# B&R Automation Studio project AriesV2
Automation Studio 4.2.7.54 SP; technology packages: mapp 1.60.1, TextSystem 

## Configuration Config_3500HS

CPU X20CP1301, AutomationRuntime D4.24, Build 4.1.2, Vc V4.24.1, Safety 1.9

### Task classes (Cpu.sw)
```
Cyclic#1 (cycle 2000 us, tolerance 0 us):
  runFirst <- Libraries.wbrServices.InitSP.runFirst.prg (BuildOptions=-D "str(x)=#x" -D AS_PROJ=str($(AS_PROJECT_NAME)) -D AS_CFG=str($(AS_CONFIGURATION)) -D "AS_VERS=str($(AS_VERSION))" -D "AS_USER=str($(AS_USER_NAME))" -D "AS_CMPNY=str($(AS_COMPANY_NAME))")
  ForceIO1 <- HMI.ForceIO.prg
  ControlLog <- Application.Master.ControlLogic.prg
  Valves <- Application.Dispense.Valves.prg
  ForceIO <- HMI.ForceIO.prg
Cyclic#8 (cycle 24000 us, tolerance 48000 us):
  wbrService <- Libraries.wbrServices.Cyclic.wbrService.prg
  HMITableMa <- HMI.HMITableManager.prg
  Recipe_Han <- Auxiliary_Services_Control.Recipe_Handling.prg  // Call functions that manage structures pertaining to params
  hmilogic <- HMI.hmilogic.prg
  ComLogger <- Auxiliary_Services_Control.ComLogger.prg [disabled]
  File_Handl <- Auxiliary_Services_Control.File_Handling.prg
DataObjects: ethIPcon
VcDataObjects: VisuW1 <- HMI.VisuW1.dob
Binaries: TCData, vccpwd, vccbtn, vcpdvnc, arialbd, vcmgr, vctcal, vcfile, vccnum, vcfntttf, vcgclass, vcbclass, vccshape, vccstr, vccalarm, vccscale, arial, vcalarm, vcdsloc, vcchtml, vccdt, vccbmp, vcshared, vcxml, vccurl, vcrt, vcctext, vcnet, vcclbox, vcdsint, vcpdsw, vccovl, vccline, VisuW101, VisuW102, VisuW103, vera, vccgauge, vcpfx20, TC, Data_Log, MAPP_Alm, MAPP_Rec, MAPP_Web, MAPP_File, MAPP_Cfg, iomap, asfw, sysconf, ashwd, arconfig, Alarm, vcctrend, vccpopup, vccddbox, vccpiech, vcpkat, verabd, Visu, Visu02, Visu03, Visu01, Axes, Config_1, MAPP_Com, Recipe, File_Mgmt, vccslider, Acp10Map1, User, Role, Data, Config, VisuW03, VisuW02, VisuW01, acp10cfg, Acp10map, Acp10sys, vcpfar00
Libraries: wbrsprintf, FileIO, AsXml, standard, runtime, astime, brsystem, sys_lib, AsANSL, AsARCfg, AsBrMath, AsBrStr, DataObj, AsTCP, AsUDP, AsUSB, MpCom, MpAlarm, MpFile, MpRecipe, MpWebXs, AsArSdm, AsIecCon, operator, AsIOTime, AsMem, AsArLog, AsArProf, MTBasics, MTTypes, MTFilter, jgLibC, MTData, ArTextSys, AsICMP, bglibasWBR, MAPPSuppor, wbrFltUtil, wbrListSvc, wbrLogSvc, wbrMemSvc, wbrPingSvc, libValve, libAS52XX, vcresman, arsvcreg, ashw, AsMbTCP, AsSafety, powerlnk
```

### Hardware
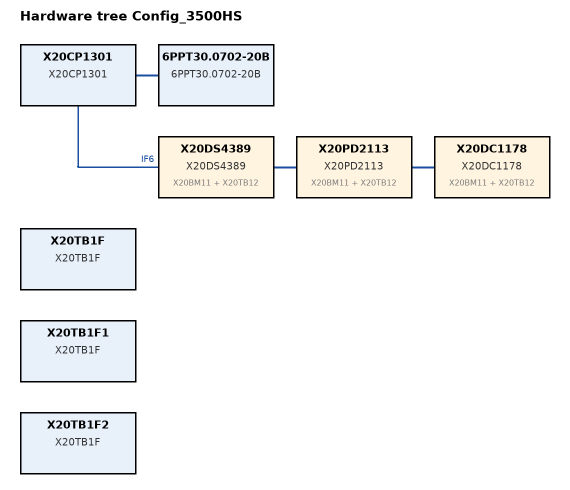
```
6PPT30.0702-20B : 6PPT30.0702-20B v1.1.0.0 (LastFrozenVersion=1.1.0.0)  [ETH1 -> X20CP1301.IF2 (NodeNumber=1)]
  Terminal = true
  Startmode = 1
  Mode = Manual
  InternetAddress = 192.168.10.20
  DefaultGateway = 192.168.10.10
  Subnetmask = 255.255.255.0
  Hostname = t30_panel
  Displaybrightness = 90
  SelectedFavoriteVNC = 192.168.10.10:5900
  PasswordVNC = 
  Favorites_Web1 = 192.168.10.10/SDM
  Favorites_Web2 = 192.168.10.10/MAPP
  USBmemoryshare = 0
  Usermemoryshare = 0
  PasswordCIFS = 
  PasswordService = 
  PPTImage = PPT_30_V1.1.0
  VncVcObjectName = VisuW1
  VncKeyMappingFile = VC\6PPT30.070.dis
  VncMaxConnections = 2
  VncRefreshRate = 300
X20BM11 : X20BM11 v1.0.0.0  [X2X1 -> X20CP1301.IF6]
X20BM11a : X20BM11 v1.0.0.0  [X2X1 -> X20BM11.X2X2]
X20BM11b : X20BM11 v1.0.0.0  [X2X1 -> X20BM11a.X2X2]
X20CP1301 : X20CP1301 v1.0.4.0  [X1 -> X1.SL; X2 -> X2.SL; X3 -> X3.SL]
  Module X1 (Type=X1, Virtual=true, Version=1.0.0.0)
    Connection (Connector=SS1, TargetModule=X20TB1F, TargetConnector=SS)
    Connection (Connector=SL, TargetModule=X20CP1301, TargetConnector=X1)
  Module X2 (Type=X2, Virtual=true, Version=1.0.0.0)
    Connection (Connector=SS1, TargetModule=X20TB1F1, TargetConnector=SS)
    Connection (Connector=SL, TargetModule=X20CP1301, TargetConnector=X2)
  Module X3 (Type=X3, Virtual=true, Version=1.0.0.0)
    Connection (Connector=SS1, TargetModule=X20TB1F2, TargetConnector=SS)
    Connection (Connector=SL, TargetModule=X20CP1301, TargetConnector=X3)
  Connector IF2:
    ActivateDevice = 1
    HostName = cp1382
    Mode = Manual
    InternetAddress = 192.168.10.10
    SubnetMask = 255.255.255.0
    InaNodeNumber = 1
  Connector IF6:
    CycleTime = 1000
  UserRamSize = 9000
  RemMemSize = 6000
  PermanentPvSize = 6000
  VolatileGlobalPvSize = 200000
  RebootPowerfail = 2
  TimerDeviceType = SWIOTIMER
  TaskClassIdleTime = 8000
  Cyclic1Duration = 2000
  Cyclic1Tolerance = 0
  Cyclic1Input = 1
  Cyclic1Output = 1
  Cyclic2Duration = 10000
  Cyclic2Tolerance = 1000000
  Cyclic3Duration = 10000
  Cyclic3Tolerance = 5000000
  Cyclic4Duration = 100000
  Cyclic4Tolerance = 100000
  Cyclic5Duration = 200000
  Cyclic5Tolerance = 200000
  Cyclic6Duration = 500000
  Cyclic6Tolerance = 500000
  Cyclic7Duration = 1000000
  Cyclic7Tolerance = 1000000
  Cyclic8Duration = 24000
  Cyclic8Tolerance = 48000
  FileDevice1
  FileDeviceName1 = ROOT
  FileDevicePath1 = F:\
  FileDevice2
  FileDeviceName2 = Recipe
  FileDevicePath2 = F:\AS_Data\Recipe
  FileDevice3
  FileDeviceName3 = Config
  FileDevicePath3 = F:\AS_Data\Config
  FtpUser1
  FtpUsername1 = user
  FtpUserPassword1 = LsodGR3jeFK3pzrFw1H5+czzepg0YTVl3svctHEKl8w=
  FtpUserSalt1 = HHFLDaL4
  FTPAccessRight1 = 0
  FtpUser2
  FtpUsername2 = admin
  FtpUserPassword2 = ohx/+BSKxELE8VtAzHGH48r+NF8pZu2EVGO55B1GtgA=
  FtpUserSalt2 = HlYZIA1j
  FTPPath2 = 5
  FTPAccessRight2 = 0
  SystemTick = 2000
X20DC1178 : X20DC1178 v1.0.0.1  [SS1 -> X20TB12b.SS; SL -> X20BM11b.SL1]
  Supervision = off
  CounterStd01 = 16Bit
  ClockrateSSI = 125kHz
  DataFormatSSI = gray
  ValidBitLengthSSI = 12
  CycleSelect = 50us
  MonoflopSSI = HIGH
  BrokenWireConfig = off
X20DS4389 : X20DS4389 v1.2.0.0  [SS1 -> X20TB12a.SS; SL -> X20BM11.SL1]
  Supervision = off
  Channel01Config = inputInv
  Channel02Config = inputInv
  Channel03Config = outputPush
  Channel04Config = outputPush
  Channel05Config = inputInv
  Channel06Config = inputInv
  Channel07Config = outputPush
  Channel08Config = outputPush
  DirectIOControlConfig = on
  EdgeDetectEnable = on
  EdgeDetectUnit01Master = 2
  EdgeDetectUnit01Slave = 18
  EdgeDetectUnit01EnableDifference = 32bit
  EdgeDetectUnit02Master = 18
  EdgeDetectUnit02Slave = 2
  EdgeDetectUnit02EnableDifference = 32bit
  EdgeDetectUnit03Master = 3
  EdgeDetectUnit03Slave = 19
  EdgeDetectUnit03EnableDifference = 32bit
  EdgeDetectUnit04Master = 19
  EdgeDetectUnit04Slave = 3
  EdgeDetectUnit04EnableDifference = 32bit
  EdgeGenerateEnable = on
  EdgeGenOutputUpdateCycle = SOAIEOP
  EdgeGenerateUnit01Enable = on
  EdgeGenUnit01TimeStamps = 1elem
  EdgeGenUnit01TimeFormat = 32bit
  EdgeGenUnit01OffsetFormat = 32bit
  EdgeGenUnit01OffsetFormat01 = cyclic
  EdgeGenUnit01Edge01Enable = on
  EdgeGenUnit01Edge01Channel = 2
  EdgeGenUnit01Edge02Enable = on
  EdgeGenerateUnit02Enable = on
  EdgeGenUnit02TimeStamps = 1elem
  EdgeGenUnit02TimeFormat = 32bit
  EdgeGenUnit02OffsetFormat = 32bit
  EdgeGenUnit02OffsetFormat01 = cyclic
  EdgeGenUnit02Edge01Enable = on
  EdgeGenUnit02Edge01Channel = 3
  EdgeGenUnit02Edge02Enable = on
  EdgeGenUnit01Edge02Channel = 18
  EdgeGenUnit02Edge02Channel = 19
  DirectIOInputs = on
X20PD2113 : X20PD2113 v1.0.2.0  [SS1 -> X20TB12.SS; SL -> X20BM11a.SL1]
X20TB12 : X20TB12 v1.0.0.0
X20TB12a : X20TB12 v1.0.0.0
X20TB12b : X20TB12 v1.0.0.0
X20TB1F : X20TB1F v1.0.0.0
X20TB1F1 : X20TB1F v1.0.0.0
X20TB1F2 : X20TB1F v1.0.0.0
```

### IoMap.iom - X20CP1301/IoMap.iom
```iecst
VAR_CONFIG
	Cyclic#1.ControlIO.iTargetPiP AT %IX."X1".DigitalInput01;
	Cyclic#1.ControlIO.iReservoirLevel AT %IX."X1".DigitalInput02;
	Cyclic#1.ControlIO.iRunCmd AT %IX."X1".DigitalInput03;
	Cyclic#1.StatusIO.iClearError AT %IX."X1".DigitalInput04;
	Cyclic#1.CureIO.iUVCuringChannelOK[0] AT %IX."X2".DigitalInput01;
	Cyclic#1.CureIO.iUVCuringChannelOK[1] AT %IX."X2".DigitalInput02;
	Cyclic#1.StatusIO.iProcessStopRelay[0] AT %IX."X2".DigitalInput03;
	Cyclic#1.StatusIO.iProcessStopRelay[1] AT %IX."X2".DigitalInput04;
	Cyclic#1.ControlIO.iX2XNettime AT %ID."X20CP1301".IF6.Nettime;
	Cyclic#1.ControlIO.iEncoderValue AT %IW."X20DC1178".Encoder01;
	Cyclic#1.StatusIO.Encoder.CycleTimeViolation.iErrorStatus AT %IX."X20DC1178".EncoderCycleTimeViolation;
	Cyclic#1.StatusIO.Encoder.DataError.iErrorStatus AT %IX."X20DC1178".EncoderDataError;
	Cyclic#1.StatusIO.Encoder.CycleTimeViolation.oQuitError AT %QX."X20DC1178".EncoderQuitCycleTimeViolation;
	Cyclic#1.StatusIO.Encoder.DataError.oQuitError AT %QX."X20DC1178".EncoderQuitDataError;
	Cyclic#1.StatusIO.Encoder.iPowerSupply[0] AT %IX."X20DC1178".PowerSupply01;
	Cyclic#1.StatusIO.Encoder.iPowerSupply[1] AT %IX."X20DC1178".PowerSupply02;
	Cyclic#1.ValveIO[0].iValveReady AT %IX."X20DS4389".DigitalInput01 INVERSE;
	Cyclic#1.ValveIO[1].iValveReady AT %IX."X20DS4389".DigitalInput02 INVERSE;
	Cyclic#1.ValveIO[0].EdgeGen.iDiffTime[0] AT %ID."X20DS4389".EdgeDetect01Difference1;
	Cyclic#1.ValveIO[0].EdgeGen.iDiffTime[1] AT %ID."X20DS4389".EdgeDetect02Difference1;
	Cyclic#1.ValveIO[0].EdgeGen.oEnableEdgeGen AT %QX."X20DS4389".EdgeGen01Enable;
	Cyclic#1.ValveIO[0].EdgeGen.iEdgeGenReadbackEnabled AT %IX."X20DS4389".EdgeGen01EnableReadback;
	Cyclic#1.ValveIO[0].EdgeGen.oEdgeGenOffset AT %QD."X20DS4389".EdgeGen01Offset1;
	Cyclic#1.ValveIO[0].EdgeGen.oEdgeGenSequence AT %QB."X20DS4389".EdgeGen01Sequence;
	Cyclic#1.ValveIO[0].EdgeGen.oEdgeGenTimestamp AT %QD."X20DS4389".EdgeGen01Timestamp1;
	Cyclic#1.ValveIO[1].EdgeGen.oEnableEdgeGen AT %QX."X20DS4389".EdgeGen02Enable;
	Cyclic#1.ValveIO[1].EdgeGen.iEdgeGenReadbackEnabled AT %IX."X20DS4389".EdgeGen02EnableReadback;
	Cyclic#1.ValveIO[1].EdgeGen.oEdgeGenOffset AT %QD."X20DS4389".EdgeGen02Offset1;
	Cyclic#1.ValveIO[1].EdgeGen.oEdgeGenSequence AT %QB."X20DS4389".EdgeGen02Sequence;
	Cyclic#1.ValveIO[1].EdgeGen.oEdgeGenTimestamp AT %QD."X20DS4389".EdgeGen02Timestamp1;
	Cyclic#1.CureIO.oUVCureChannel[0] AT %QX."X3".DigitalOutput01;
	Cyclic#1.CureIO.oUVCureChannel[1] AT %QX."X3".DigitalOutput02;
	Cyclic#1.StatusIO.oRunningReady AT %QX."X3".DigitalOutput04;
	Cyclic#1.StatusIO.oSystemNeedsAttention AT %QX."X3".DigitalOutput05;
	Cyclic#1.ControlIO.oTargetPresent AT %QX."X3".DigitalOutput06;
	Cyclic#1.ControlIO.Inspection.oInspectionGood AT %QX."X3".DigitalOutput07;
	Cyclic#1.ControlIO.Inspection.oInspectionValid AT %QX."X3".DigitalOutput08;
	Cyclic#1.StatusIO.oStatusColor.Red AT %QX."X3".DigitalOutput09;
	Cyclic#1.StatusIO.oStatusColor.Green AT %QX."X3".DigitalOutput10;
	Cyclic#1.StatusIO.oStatusColor.Blue AT %QX."X3".DigitalOutput11;
END_VAR
```

### Data_Log.mpdatarecorder - X20CP1301/mapp/Data_Log.mpdatarecorder
```
Element Data_Log_MpLink (Type=mpdatarecorder)
  DataRecorder:
    MaxNumberOfFiles = 15
    DecimalDigits = 3
    SaveInterval = 60000
    PowerFailSafe = FALSE
    DecimalMark = .
    OverwriteOldestFile = TRUE
```

## Configuration Config_Deployment

### Task classes (Cpu.sw)
```
Cyclic#1 (cycle 4000 us, tolerance 0 us):
  ForceIO <- HMI.ForceIO.prg
  Creaser <- Application.Creaser.prg
  ForceIO1 <- HMI.ForceIO.prg
Cyclic#8 (cycle 8000 us, tolerance 30000000 us):
  LineContro <- MotionControl.LineControl.prg
  HMI_Alarms <- HMI.HMI_Alarms.prg
  Recipe_Han <- Auxiliary_Services_Control.Recipe_Handling.prg
  hmilogic <- HMI.hmilogic.prg
  HMITableMa <- HMI.HMITableManager.prg
  File_Handl <- Auxiliary_Services_Control.File_Handling.prg
  ComLogger <- Auxiliary_Services_Control.ComLogger.prg
DataObjects: Acp10sys, ethIPcon
NcDataObjects: acp10etxen <- acp10etxen.dob, Axisa <- Axisobj.Axisa.dob, Axisi <- Axisobj.Axisi.dob
VcDataObjects: Visup <- HMI.Visup.dob
Binaries: vcfntttf, vccbmp, vcshared, vccscale, vcpdvnc, Visup01, vcfile, vccpwd, arial, Visup03, vcmgr, vcxml, vcdsint, vccbtn, vcdsloc, vccalarm, vccovl, vcpfx20, vccline, vcctext, vcalarm, vcbclass, vcgclass, udbdef, vcrt, vccnum, vccstr, vccddbox, arialbd, vera, vccshape, vcpdsw, vccpopup, Visup02, vccurl, vcnet, arsvcreg, TCData, vcchtml, vctcal, vccdt, vcpkat, vcclbox, Data_Log, MAPP_Alm, MAPP_Rec, Alarm, MAPP_Web, ashwd, arconfig, MAPP_File, Config, asfw, sysconf, TC, MAPP_Cfg, iomap, acp10cfg, Acp10map, vcpfar00, Visu102, Visu101, Visu103, VisuW101, vcctrend, vccpiech, verabd, Visu, Visu02, Visu03, Visu01, Axes, Config_1, MAPP_Com, Recipe, File_Mgmt, vccslider, Acp10Map1, User, Role, Data, VisuW03, VisuW02, VisuW01, vccgauge, VisuW103, VisuW102
Libraries: FileIO, AsXml, standard, runtime, astime, brsystem, sys_lib, AsANSL, AsARCfg, AsBrMath, AsBrStr, DataObj, AsTCP, AsUDP, AsUSB, AsArSdm, AsIecCon, operator, AsIOTime, AsMem, AsArLog, AsArProf, AsICMP, Acp10man, Acp10par, NcGlobal, Acp10_MC, MpAxis, MpCom, wbrsprintf, wbrPingSvc, wbrMemSvc, wbrLogSvc, wbrListSvc, wbrFltUtil, MpWebXs, MpRecipe, MpFile, MpAlarm, MAPPSuppor, jgLibC, bglibasWBR, Acp10sim, ArTextSys, vcresman, powerlnk, ashw, MTTypes, AsMbTCP, AsSafety, MTData
```

### Hardware
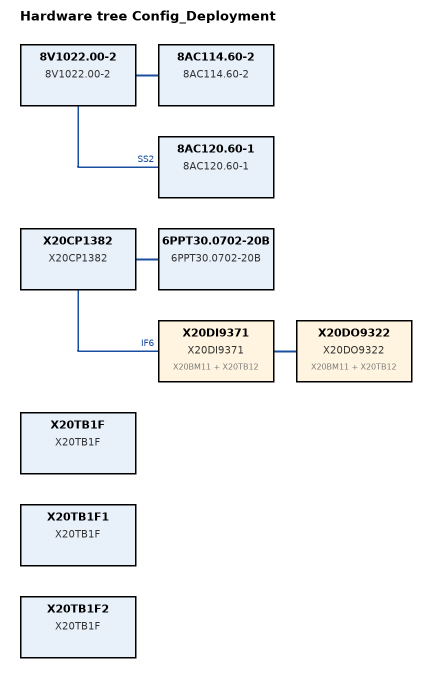
```
6PPT30.0702-20B : 6PPT30.0702-20B v1.1.0.0  [ETH1 -> X20CP1382.IF2 (NodeNumber=1)]
  Terminal = true
  Startmode = 1
  ShowBootlogoVNC = 1
  Mode = Manual
  InternetAddress = 192.168.10.20
  DefaultGateway = 192.168.10.1
  Subnetmask = 255.255.255.0
  Displaybrightness = 75
  SelectedFavoriteVNC = 192.168.10.10
  Favorites_VNC1 = 192.168.10.10
  PasswordVNC = 
  PasswordCIFS = 
  PasswordService = 
  PPTImage = PPT_30_V1.1.1
  VncRefreshRate = 200
8AC114.60-2 : 8AC114.60-2 v1.0.0.8  [SS -> 8V1022.00-2.SS1; PLK1 -> X20CP1382.IF3 (NodeNumber=2)]
8AC120.60-1 : 8AC120.60-1 v1.0.0.2  [SS -> 8V1022.00-2.SS2]
8V1022.00-2 : 8V1022.00-2 v1.0.0.2
  AxisIsPeriodic_r1 = on
  BothEndSwitchesAreNormallyOpen_r1 = on
  QuickStopIsNormallyOpen_r1 = on
X20BM11 : X20BM11 v1.0.0.1  [X2X1 -> X20CP1382.IF6]
X20BM11a : X20BM11 v1.0.0.1  [X2X1 -> X20BM11.X2X2]
X20CP1382 : X20CP1382 v1.3.2.0  [X1 -> X1.SL; X2 -> X2.SL; X3 -> X3.SL]
  Module X1 (Type=X1, Virtual=true, Version=1.0.0.0)
    Connection (Connector=SS1, TargetModule=X20TB1F, TargetConnector=SS)
    Connection (Connector=SL, TargetModule=X20CP1382, TargetConnector=X1)
  Module X2 (Type=X2, Virtual=true, Version=1.0.0.0)
    Connection (Connector=SS1, TargetModule=X20TB1F1, TargetConnector=SS)
    Connection (Connector=SL, TargetModule=X20CP1382, TargetConnector=X2)
  Module X3 (Type=X3, Virtual=true, Version=1.0.0.0)
    Connection (Connector=SS1, TargetModule=X20TB1F2, TargetConnector=SS)
    Connection (Connector=SL, TargetModule=X20CP1382, TargetConnector=X3)
  Connector IF2:
    ActivateDevice = 1
    HostName = x20cpu
    Mode = Manual
    InternetAddress = 192.168.10.10
    SubnetMask = 255.255.255.0
    InaNodeNumber = 0
    Vnc1
    VncVcObjectName1 = Visup
    VncKeyMappingFile1 = VC\PS2-Keyboard4.dis
    VncRefreshRate1 = 200
  Connector IF3:
    CycleTime = 4000
  Connector IF6:
    CycleTime = 4000
  ConfigurationID = AriesV2_Config_Test
  UserPartitionSize = 256
  UserRamSize = 5000
  RemMemSize = 25000
  PermanentPvSize = 15000
  VolatileGlobalPvSize = 300000
  RebootReset = 2
  RebootPowerfail = 2
  TimerDeviceType = EPLX2X
  TimerDevice = X20CP1382.IF3
  TaskClassIdleTime = 8000
  Cyclic1Duration = 4000
  Cyclic1Tolerance = 0
  Cyclic2Duration = 16000
  Cyclic2Tolerance = 16000
  Cyclic3Duration = 48000
  Cyclic3Tolerance = 48000
  Cyclic4Duration = 96000
  Cyclic4Tolerance = 96000
  Cyclic5Duration = 200000
  Cyclic5Tolerance = 200000
  Cyclic6Duration = 496000
  Cyclic6Tolerance = 496000
  Cyclic7Duration = 1000000
  Cyclic7Tolerance = 1000000
  Cyclic8Duration = 8000
  Cyclic8Tolerance = 30000000
  FileDevice1
  FileDeviceName1 = ROOT
  FileDevicePath1 = F:\
  FileDevice2
  FileDeviceName2 = Config
  FileDevicePath2 = F:\Config
  FileDevice3
  FileDeviceName3 = Recipe
  FileDevicePath3 = F:\Recipe
  FileDevice4
  FileDeviceName4 = Process
  FileDevicePath4 = F:\Process
  FtpUser1
  FtpUsername1 = admin
  FtpUserPassword1 = tXcQUdKIsoY/H/jtKSqzHLRzyWbO/eZFb+QmJVs8vuM=
  FtpUserSalt1 = fFlgpUU6
  FTPAccessRight1 = 0
  FTPdevice1 = ALL
  FtpUser2
  FtpUsername2 = user
  FtpUserPassword2 = M/sBBWLbPcMSL0ECBo9+NNWk5QFExAfaSSh+paOlJpQ=
  FtpUserSalt2 = diDYFxUT
  FTPAccessRight2 = 0
  FTPMSpath2 = /
X20DI9371 : X20DI9371 v1.0.1.3  [SS1 -> X20TB12.SS; SL -> X20BM11.SL1]
  Supervision = off
X20DO9322 : X20DO9322 v1.0.3.0  [SS1 -> X20TB12a.SS; SL -> X20BM11a.SL1]
  Supervision = off
X20TB12 : X20TB12 v1.0.0.0
X20TB12a : X20TB12 v1.0.0.0
X20TB1F : X20TB1F v1.0.0.0
X20TB1F1 : X20TB1F v1.0.0.0
X20TB1F2 : X20TB1F v1.0.0.0
```

### Config.mpaxisbasic - X20CP1382/mapp/Config.mpaxisbasic
```
Element FeedAxis_MpLink (Type=mpaxisbasic)
  AxisConfiguration = AxisWithConfiguration
    Axis:
      MeasurementUnit = 1
      MeasurementResolution = 0.001
      PeriodSettings:
        Period = 125.664
      MovementLimits:
        VelocityPositive = 10000.0
        VelocityNegative = 10000.0
        Acceleration = 10000.0
        Deceleration = 10000.0
        PositionErrorStopLimit = 1
    Drive:
      Gearbox:
        Input = 5
      Transformation:
        ReferenceDistance = 125.664
      Controller:
        Speed:
          ProportionalGain = 1.75
          IntegralTime = 1
        LoopFilters:
          [0]
          [1]
          [2]
```

## Configuration Config_Test

CPU X20CP1382, AutomationRuntime B4.26, Build 4.1.2, Vc V4.26.3, Safety 0.0

CPU X20CP1584, AutomationRuntime B4.26, Build 4.1.2, Vc not used, Safety 1.5

### Task classes (Cpu.sw)
```
Cyclic#1 (cycle 8000 us, tolerance 0 us):
  ForceIO <- HMI.ForceIO.prg [disabled]
  Creaser <- Application.Creaser.prg
  ForceIO1 <- HMI.ForceIO.prg [disabled]
DataObjects: ethIPcon
NcDataObjects: acp10etxen <- acp10etxen.dob, Axisa <- Axisobj.Axisa.dob, Axisi <- Axisobj.Axisi.dob
Binaries: TCData, Acp10sys, udbdef, Alarm, ashwd, asfw, MAPP_Cfg, MAPP_File, MAPP_Web, MAPP_Rec, MAPP_Alm, Data_Log, arconfig, sysconf, iomap, Config, acp10cfg, Acp10map, vcpdvnc, vcmgr, vctcal, vcnet, VisuW101, vcpfx20, vcctrend, vccpopup, vccddbox, vccpiech, vcpkat, verabd, Visu, Visu02, Visu03, Visu01, Axes, Config_1, MAPP_Com, Recipe, File_Mgmt, vccslider, Acp10Map1, User, Role, Data, VisuW03, VisuW02, VisuW01, vcpfar00, TC, vccgauge, vera, VisuW103, VisuW102, vccline, vccovl, vcpdsw, vcdsint, vcclbox, vcctext, vcrt, vccurl, vcxml, vcshared, vccbmp, vccdt, vcchtml, vcdsloc, vcalarm, arial, vccscale, vccalarm, vccstr, vccshape, vcbclass, vcgclass, vcfntttf, vccnum, vcfile, arialbd, vccbtn, vccpwd
Libraries: FileIO, AsXml, standard, runtime, astime, brsystem, sys_lib, AsANSL, AsARCfg, AsBrMath, AsBrStr, DataObj, AsTCP, AsUDP, AsUSB, AsArSdm, AsIecCon, operator, AsIOTime, AsMem, AsArLog, AsArProf, AsICMP, powerlnk, Acp10man, Acp10par, NcGlobal, Acp10_MC, MpAxis, MpCom, wbrsprintf, wbrPingSvc, wbrMemSvc, wbrLogSvc, wbrListSvc, wbrFltUtil, MpWebXs, MpRecipe, MpFile, MpAlarm, MAPPSuppor, jgLibC, bglibasWBR, arsvcreg, ashw, AsMbTCP, AsSafety, vcresman
```

### Task classes (Cpu.sw)
```
DataObjects: ethIPcon
Binaries: TCData, Alarm, ashwd, asfw, MAPP_Cfg, MAPP_File, MAPP_Web, MAPP_Rec, MAPP_Alm, Data_Log, arconfig, sysconf, iomap, vcpdvnc, vcmgr, vctcal, vcnet, VisuW101, vcpfx20, vcctrend, vccpopup, vccddbox, vccpiech, vcpkat, verabd, Visu, Visu02, Visu03, Visu01, Axes, Config_1, MAPP_Com, Recipe, File_Mgmt, vccslider, Acp10Map1, User, Role, Data, Config, VisuW03, VisuW02, VisuW01, acp10cfg, Acp10map, Acp10sys, vcpfar00, TC, vccgauge, vera, VisuW103, VisuW102, vccline, vccovl, vcpdsw, vcdsint, vcclbox, vcctext, vcrt, vccurl, vcxml, vcshared, vccbmp, vccdt, vcchtml, vcdsloc, vcalarm, arial, vccscale, vccalarm, vccstr, vccshape, vcbclass, vcgclass, vcfntttf, vccnum, vcfile, arialbd, vccbtn, vccpwd
Libraries: FileIO, AsXml, standard, runtime, astime, brsystem, sys_lib, AsANSL, AsARCfg, AsBrMath, AsBrStr, DataObj, AsTCP, AsUDP, AsUSB, AsArSdm, AsIecCon, operator, AsIOTime, AsMem, AsArLog, AsArProf, AsICMP, arsvcreg, ashw, AsMbTCP, AsSafety, powerlnk, vcresman
```

### Hardware
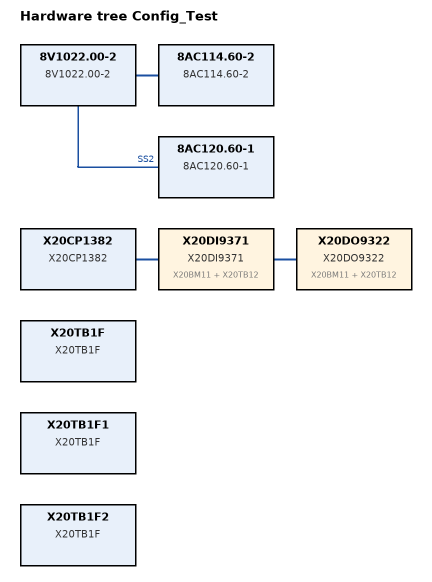
```
8AC114.60-2 : 8AC114.60-2 v1.0.0.8  [SS -> 8V1022.00-2.SS1; PLK1 -> X20CP1382.IF3 (NodeNumber=2)]
8AC120.60-1 : 8AC120.60-1 v1.0.0.2  [SS -> 8V1022.00-2.SS2]
8V1022.00-2 : 8V1022.00-2 v1.0.0.2
  AxisIsPeriodic_r1 = on
  BothEndSwitchesAreNormallyOpen_r1 = on
  QuickStopIsNormallyOpen_r1 = on
X20BM11 : X20BM11 v1.0.0.1  [X2X1 -> X20CP1382.IF6]
X20BM11a : X20BM11 v1.0.0.1  [X2X1 -> X20BM11.X2X2]
X20CP1382 : X20CP1382 v1.3.2.0  [X1 -> X1.SL; X2 -> X2.SL; X3 -> X3.SL]
  Module X1 (Type=X1, Virtual=true, Version=1.0.0.0)
    Connection (Connector=SS1, TargetModule=X20TB1F, TargetConnector=SS)
    Connection (Connector=SL, TargetModule=X20CP1382, TargetConnector=X1)
  Module X2 (Type=X2, Virtual=true, Version=1.0.0.0)
    Connection (Connector=SS1, TargetModule=X20TB1F1, TargetConnector=SS)
    Connection (Connector=SL, TargetModule=X20CP1382, TargetConnector=X2)
  Module X3 (Type=X3, Virtual=true, Version=1.0.0.0)
    Connection (Connector=SS1, TargetModule=X20TB1F2, TargetConnector=SS)
    Connection (Connector=SL, TargetModule=X20CP1382, TargetConnector=X3)
  Connector IF2:
    ActivateDevice = 1
    HostName = x20cpu
    Mode = Manual
    InternetAddress = 192.168.10.10
    SubnetMask = 255.255.255.0
    InaNodeNumber = 0
    Vnc1
    VncVcObjectName1 = Visu1
    VncKeyMappingFile1 = VC\PS2-Keyboard4.dis
    VncRefreshRate1 = 200
  Connector IF3:
    CycleTime = 8000
  Connector IF6:
    CycleTime = 8000
  ConfigurationID = AriesV2_Config_Test
  UserRamSize = 5000
  RemMemSize = 25000
  PermanentPvSize = 15000
  VolatileGlobalPvSize = 300000
  RebootReset = 2
  RebootPowerfail = 2
  TimerDeviceType = EPLX2X
  TimerDevice = X20CP1382.IF3
  TaskClassIdleTime = 8000
  Cyclic1Duration = 8000
  Cyclic1Tolerance = 0
  Cyclic2Duration = 16000
  Cyclic2Tolerance = 16000
  Cyclic3Duration = 48000
  Cyclic3Tolerance = 48000
  Cyclic4Duration = 96000
  Cyclic4Tolerance = 96000
  Cyclic5Duration = 200000
  Cyclic5Tolerance = 200000
  Cyclic6Duration = 496000
  Cyclic6Tolerance = 496000
  Cyclic7Duration = 1000000
  Cyclic7Tolerance = 1000000
  Cyclic8Duration = 8000
  Cyclic8Tolerance = 30000000
  FileDevice1
  FileDeviceName1 = ROOT
  FileDevicePath1 = F:\
  FileDevice2
  FileDeviceName2 = Config
  FileDevicePath2 = F:\Config
  FileDevice3
  FileDeviceName3 = Recipe
  FileDevicePath3 = F:\Recipe
  FileDevice4
  FileDeviceName4 = Process
  FileDevicePath4 = F:\Process
X20DI9371 : X20DI9371 v1.0.2.0  [SS1 -> X20TB12.SS; SL -> X20BM11.SL1]
  Supervision = off
X20DO9322 : X20DO9322 v1.0.3.0  [SS1 -> X20TB12a.SS; SL -> X20BM11a.SL1]
  Supervision = off
X20TB12 : X20TB12 v1.0.0.0
X20TB12a : X20TB12 v1.0.0.0
X20TB1F : X20TB1F v1.0.0.0
X20TB1F1 : X20TB1F v1.0.0.0
X20TB1F2 : X20TB1F v1.0.0.0
```

### Cpu.per - X20CP1382/Cpu.per
```iecst
VAR_CONFIG
	gRecipeName AT %M0; (* *)
	gConfigName AT %M256; (* *)
	gStatistics AT %M512; (* *)
	gRecCfg AT %M600; (* *)
END_VAR
```

### Acp10map.ncm - X20CP1584/Motion/Acp10map.ncm
```
NcMapping (NcSwId=Acp10)
  NcObject Axis (ModuleId=8V1045.00-2, Type=ncAXIS, Channel=1, AcoposSimulation=Off, InitParameter=Axisi, AcoposParameter=Axisa, AdditionalData=PLCopen_ModPos="1000,1" , Disabled=FALSE, ModuleDisabled=FALSE)
  NcObject 8V1045.00-2_ncV_AXIS1 (ModuleId=8V1045.00-2, Type=ncV_AXIS, Channel=1, Disabled=TRUE, ModuleDisabled=FALSE)
```

### Config.mpaxisbasic - X20CP1584/mapp/Config.mpaxisbasic
```
Element FeedAxis_MpLink (Type=mpaxisbasic)
  AxisConfiguration = AxisWithConfiguration
    Axis:
      MeasurementUnit = 1
      MeasurementResolution = 0.001
      PeriodSettings:
        Period = 125.664
    Drive:
      Gearbox:
        Input = 5
      Transformation:
        ReferenceDistance = 125.664
      Controller:
        LoopFilters:
          [0]
          [1]
          [2]
```

### Cpu.per - X20CP1585/Cpu.per
```iecst
VAR_CONFIG
	gRecipeName AT %M0; (* *)
	gConfigName AT %M256; (* *)
	gRecCfg AT %M512; (* *)
END_VAR
```

## Logical view

Binary libraries used (declarations not repeated): operator, runtime, astime, AsIecCon, FileIO, AsXml, standard, brsystem, sys_lib, AsANSL, AsARCfg, AsBrMath, AsBrStr, DataObj, AsTCP, AsUDP, AsUSB, AsArSdm, AsIOTime, AsMem, AsArLog, AsArProf, MTTypes, jgLibC, MTData, AsICMP, MpCom, MpAxis, MpWebXs, MpRecipe, MpAlarm, MpFile 1.20.5, ArTextSys 0.16.0, Acp10man 3.16.1, Acp10par, NcGlobal, Acp10sim 3.16.1, Acp10_MC 3.16.1, libValve

- Hernon SureShot Controller Job 3647_GD_rev3.xlsx (binary file, 432008 bytes)
### Global.var
```iecst
VAR CONSTANT
	FORCEIO_ACCESS_LEVEL : UINT := 1;
	CONFIG_ACCESS_LEVEL : UINT := 2;
	RECIPE_ACCESS_LEVEL : UINT := 1;
	DEFINE_MENU_L_HIDE_TIMEOUT_MS : UDINT := 7000;
	DEFINE_MENU_R_HIDE_TIMEOUT_MS : UDINT := 7000;
	DEFINE_HMI_SPLASHSCREEN_TO_MS : UDINT := 5000;
	MAX_IDX_TOTAL_RECIPES : UINT := 100;
	DEFINE_LOGIN_TO : REAL := 600;
END_VAR
(*Insert your comment here.*)
VAR CONSTANT
	MAX_IDX_CREASES : UDINT := 19;
END_VAR
(*Insert your comment here.*)
(*Insert your comment here.*)
VAR RETAIN
	gRecCfg : Global_Par_typ;
END_VAR
VAR
	gAcknowledge : Machine_Alarms_typ;
	gAlarms : Machine_Alarms_typ;
	gMachineName : {REDUND_UNREPLICABLE} STRING[80] := 'Aries';
	gProjectDate : {REDUND_UNREPLICABLE} STRING[80] := '10. April 2017';
	gVersion : {REDUND_UNREPLICABLE} STRING[80] := 'R777';
END_VAR
(*Insert your comment here.*)
VAR
	Axis1 : ACP10AXIS_typ;
	AxisControl : MpAxisBasic;
	AxisPar : MpAxisBasicParType;
	Alarm_Feed : MpAlarmBasicUIConnect20Type := (0);
	Alarm_Feed_UI : MpAlarmBasicUI := (0);
END_VAR
(*Insert your comment here.*)
VAR
	MachineState : AriesMachineState_Enum;
	ProcessState : CreaserPrcsState_Enum;
END_VAR
(*Insert your comment here.*)
VAR
	IO : AriesIOPoints_typ;
	IO_LastCycle : AriesIOPoints_typ;
END_VAR
(*Insert your comment here.*)
VAR
	AppAlarms : MpAlarmBasicUIConnect20Type;
	AppAlarms_FBK : MpAlarmBasic;
	AppAlarms_UI : USINT;
END_VAR
(*Insert your comment here.*)
VAR RETAIN
	gStatistics : Global_Statistics_typ;
END_VAR
(*Insert your comment here.*)
VAR
	gAlarmResetRequested : BOOL;
	StartUIButton_Hide : USINT;
	StopUIButton_Hide : USINT;
	BoardEjectUIButton_Hide : USINT;
	iManualBoardEject : BOOL;
	iMachineErrorReset : BOOL;
	iStartCommand : BOOL;
	iSoftStopCommand : BOOL;
	gSimulateMachine : BOOL;
END_VAR
(*Insert your comment here.*)
VAR CONSTANT
	DEFINE_MM_ROLLER_REV : REAL := 125.664;
END_VAR
VAR
	delta_Board_Position : REAL;
	RollerPos_LastCycle : REAL;
	RollerPos_ThisCycle : REAL;
	Current_Board_Position : REAL;
	Latch_Board_Length : REAL;
	Current_Crease_Section_Length : REAL;
END_VAR
(*Insert your comment here.*)
(*Insert your comment here.*)
```

### Machine.typ
```iecst
TYPE
	CreaserPrcsState_Enum :
		( (*Make sure the indices entered below line up with the VC texts displayed on the UI*)
		PRCS_STATE_INIT := 0,
		PRCS_STATE_READY := 1,
		PRCS_STATE_FEED_BOARD := 2,
		PRCS_STATE_MOVE_CREASE := 3,
		PRCS_STATE_CREASE := 4,
		PRCS_STATE_MOVE_CREASE_WIDTH := 5,
		PRCS_STATE_ERROR := 6,
		PRCS_STATE_EJECT_FINISHED_BOARD := 7,
		PRCS_STATE_SOFT_STOP := 8,
		PRCS_STATE_MOVE_PHOTOEYE_OFFSET := 9
		);
	AriesMachineState_Enum :
		( (*Make sure the indices entered below line up with the VC texts displayed on the UI*)
		MACHINE_STATE_INIT := 0,
		MACHINE_STATE_IDLE := 1,
		MACHINE_STATE_RUNNING := 2,
		MACHINE_STATE_ERROR := 3,
		MACHINE_STATE_HARDWARE_INIT := 4,
		MACHINE_STATE_AXIS_POWER := 5,
		MACHINE_STATE_AXIS_HOME := 6,
		MACHINE_STATE_MANUAL_EJECT := 7
		);
END_TYPE

(*Insert your comment here.*)

TYPE
	CreaserConfig_typ : 	STRUCT
		FeedAxisAccel : REAL;
		FeedAxisDecel : REAL;
		PhotoEyeOffset : REAL;
		PreInsertSpeed : REAL;
		BoardLengthTolerance : REAL;
		CreaseInfeedDelay : REAL;
		BypassBoardLengthError : UDINT;
		PhotoEyeMeasurementOffset : REAL;
	END_STRUCT;
	AriesCreaserParams_typ : 	STRUCT
		CreaseDistance_mm : ARRAY[0..MAX_IDX_CREASES]OF REAL;
		CreaseWidth_mm : REAL;
		CreaseCount : UDINT;
		ShaftSensorEdge : UDINT;
		CreaserDirection : UDINT;
		CreaserMotorIdxLag_S : REAL;
		TotalBoardLength : REAL;
	END_STRUCT;
END_TYPE

(*Insert your comment here.*)

TYPE
	AriesIOPoints_typ : 	STRUCT
		oCreaserCCWRotation : BOOL;
		oCreaserCWRotation : BOOL;
		oBoardFeedingLight : BOOL;
		oUIIndicatorLight : BOOL;
		iSafeMachineState : BOOL;
		iCreaserShaftSensor : BOOL;
		iFiberOpticSensor : BOOL;
		iSM1Disabled : BOOL;
	END_STRUCT;
END_TYPE

(*Insert your comment here.*)

TYPE
	Machine_Alarms_typ : 	STRUCT  (*Did something fancy here- structure is copied into array for VC error texts, make sure the following numbers line up with the VC error text indices!*)
		SM1_Disabled : BOOL; (*0*)
		Unsafe_Machine_State : BOOL; (*1*)
		Fiber_Optic_Blocked_RunCmd : BOOL; (*2*)
		Creaser_Shaft_Edge_Timeout : BOOL; (*3*)
		Error_State_Unsafe_Machine : BOOL; (*4*)
		Error_State_SM1_Power : BOOL; (*5*)
		Feed_Axis_Motor_Error : BOOL; (*6*)
		Crease_Count_Greater_Max : BOOL; (*7*)
		Error_State_Process_Error : BOOL; (*8*)
		Load_Recipe : BOOL; (*9*)
		Manual_Home_Creaser_Blade : BOOL; (*10*)
		Board_Length_GT_Confgd_Amount : BOOL; (*11*)
		Board_Length_LT_Confgd_Amount : BOOL; (*12*)
		Measured_Length_GT_Configured : BOOL; (*13*)
		Measured_Length_LT_Configured : BOOL; (*14*)
		Unsaved_Recipe_Params : BOOL; (*15*)
	END_STRUCT;
	Global_Statistics_typ : 	STRUCT
		total_runtime : UDINT;
		runtime_h : UDINT;
		runtime_m : UDINT;
		runtime_s : UDINT;
		total_processed : UDINT;
		Reset : BOOL;
		total_creases : UDINT;
		Sum_Board_Travel_Lengths : REAL;
		Avg_Board_Length : REAL;
	END_STRUCT;
END_TYPE
```

### Generic_Rec_Cfg.typ
```iecst
TYPE
	HMIConfig_typ : 	STRUCT
		passwordSetup : STRING[15];
		passwordEngineer : STRING[15];
		passwordFactory : STRING[15];
		MachineLang : UDINT;
	END_STRUCT;
END_TYPE

(*Insert your comment here.*)

TYPE
	Global_Rec_typ : 	STRUCT
		MagicPrefix : UDINT;
		MagicSuffix : UDINT;
	END_STRUCT;
	Global_Cfg_typ : 	STRUCT
		MagicPrefix : UDINT;
		HMI : HMIConfig_typ;
		wbrMemService : wbrMemService_typ;
		cfgCompile : cfgCompileVersionInfo_typ;
		MagicSuffix : UDINT;
	END_STRUCT;
END_TYPE

(*Insert your comment here.*)

TYPE
	Global_Rec_Cfg_typ : 	STRUCT
		Rec : Global_Rec_typ;
		Cfg : Global_Cfg_typ;
	END_STRUCT;
	Global_RecCfg_Public_In_typ : 	STRUCT
		Copy_default_to_save : USINT;
		Copy_default_to_active : USINT;
		Copy_save_to_active : USINT;
		Copy_save_to_default : USINT;
		Copy_active_to_save : USINT;
		Copy_active_to_default : USINT;
		Copy_internal_to_default : USINT;
		FileName : STRING[255];
	END_STRUCT;
	Global_RecCfg_Public_Out_typ : 	STRUCT
		save_differs_from_active : USINT;
		default_differs_from_save : USINT;
		active_differs_from_default : USINT;
	END_STRUCT;
	Global_Rec_Cfg_Info_typ : 	STRUCT
		O : Global_RecCfg_Public_Out_typ;
		I : Global_RecCfg_Public_In_typ;
	END_STRUCT;
	Global_Rec_Cfg_IO_typ : 	STRUCT
		Rec : Global_Rec_Cfg_Info_typ;
		Cfg : Global_Rec_Cfg_Info_typ;
	END_STRUCT;
	Global_Par_typ : 	STRUCT
		save : Global_Rec_Cfg_typ;
		active : Global_Rec_Cfg_typ;
		defaultvals : Global_Rec_Cfg_typ;
		IO : Global_Rec_Cfg_IO_typ;
	END_STRUCT;
END_TYPE

(*Insert your comment here.*)
```

### Package Logical/Libraries - Global libraries

### Library Logical/Libraries/MAPPSuppor (ANSIC) - library (written/managed by J. Glisson) containing functions for ACPu err acknowledgement, HMI param table construction, HMI param table activation to the common layer
Depends on: standard, sys_lib, wbrLogSvc, ArTextSys

#### bgsprintf.h
```c
/*
File:
bgSprintf.h

About:
------
- short and limited implementation of the sprintf() function

*/
#ifndef _BG_SPRINTF_H
#define _BG_SPRINTF_H

//#include <stdarg.h>

/*
Public data types:
-----------------
*/

/*
Public functions:
-----------------
*/
int bgsprintf(char *out, const char *format, ...);

int bgsnprintf(char *out, int size, const char *format, ...);

//int bgvsprintf(char *out, const char *format, va_list args);

#endif
```

#### ActivateHMITable.c
```c
#include <bur/plctypes.h>
#ifdef __cplusplus
	extern "C"
	{
#endif
	#include "MAPPSuppor.h"
#ifdef __cplusplus
	};
#endif
#include "hmiParamList.h"
#include "ArTextSys.h"
/* TODO: Add your comment here */

REAL PVStructInfo(PVListTexts_Info_typ * p){

	UDINT val_int = 0;
	REAL val_real = 0;

	if(!p || !(p->isValid)){
		return 0;
	}else if(p->isConstant){
		return p->Const_Value;
	}

	switch(p->PVTyp){
		case 7: //UDINT
			val_int = *((UDINT *)(p->PVAdr));
			val_real = (REAL) val_int;
			break;
		case 8: //REAL
			val_real = *((REAL * )(p->PVAdr));
			break;
	}

	return val_real;

}

plcbit ActivateHMITable(DINT langIdx, UDINT pHMITable_int, UDINT pTableValues_int)
{
	hmiParamListTable_typ * pHMITable = pHMITable_int;
	HMI_Table_Data_typ * pTableValues = pTableValues_int;
	UDINT ii_entries = 0;
	UINT valtype;
	DINT dec_places;
	REAL val_min;
	REAL val_max;
	REAL val_def;
	UDINT * val_hide_int;

	BOOL val_hide_bool = 0;

	if(pTableValues->Max_Idx_Entries >= DEFINE_MAX_TABLE_ENTRIES) return 0;

	hmiParamListTableEntryFirst(pHMITable, (char *) &pTableValues->Table_Name);
	for(ii_entries = 0; ii_entries <= pTableValues->Max_Idx_Entries; ii_entries++){
		if(pTableValues->info[ii_entries].Val.Hide.isValid==1){
			if(pTableValues->info[ii_entries].Val.Hide.isPV==1){
				val_hide_int = ((UDINT *) (pTableValues->info[ii_entries].Val.Hide.PVAdr));
				val_hide_bool = (BOOL) (*val_hide_int);
			}else{
				val_hide_bool = (BOOL) pTableValues->info[ii_entries].Val.Hide.Const_Value;
			}
		}else{
			val_hide_bool = 0;
		}

		if(val_hide_bool==0 && pTableValues->info[ii_entries].Val.Param.PVAdr){
			val_min = PVStructInfo(&pTableValues->info[ii_entries].Val.Min);
			val_max = PVStructInfo(&pTableValues->info[ii_entries].Val.Max);
			val_def = PVStructInfo(&pTableValues->info[ii_entries].Val.Default);

				switch(pTableValues->info[ii_entries].Val.Param.PVTyp){
					case 7: //UDINT
						valtype=0;
						dec_places=-2; //no decimals
						break;
					case 8: //REAL
						valtype=1;
						dec_places=1;
						break;
				}

				hmiParamListTableAddEntryNext(pHMITable,
					pTableValues->info[ii_entries].Val.Param.PVAdr,
					&pTableValues->info[ii_entries].PVText[langIdx].PVTextLangSpecific,
					val_def,val_min,val_max,
					dec_places,1,0,valtype,
					&pTableValues->info[ii_entries].PVText[langIdx].PVDescLangSpecific
					);
			}
		}
	hmiParamListTableEntryLast(pHMITable);
}
```

### Package Logical/Libraries/wbrServices - Service libraries

- Program Logical/Libraries/wbrServices/Cyclic/wbrService (ANSIC) - Cyclic updates for wbrServices libraries.  Place in TC#8 (no source held here)

### Program Logical/Libraries/wbrServices/InitSP/runFirst

#### svninfo.c
```c
char *Revision      = "777";
char *Modified      = "Modified";
char *Date          = "2017/04/27 17:02:14";
char *TimeNow       = "2017/04/28 11:53:04";
char *RevRange      = "776:777";
char *Mixed         = "Mixed revision WC";
char *IsTagged      = "Not tagged";
char *URL           = "http://99.33.212.60/Internal/MarketingAlliance/trunk/software/AriesV2";
char *isInSVN       = "not versioned";
char *lockdate      = "1969/12/31 19:00:00";
```

### Program Logical/Libraries/wbrServices/TimerServices/msTimeSvc

#### msTimeSvc.c
```c
/********************************************************************
 * \copyright -- Piedmont Automation
 ********************************************************************
 * Program : msTimeSvc
 * \file :   msTimeSvc.c
 * \author : Blanton Radford
 * \date Created: May 07, 2015
 ********************************************************************
 * \brief Implementation of program msTimeSvc
 ********************************************************************/

/********************************************************************
 * COPYRIGHT -- Piedmont Automation
 ********************************************************************
 * Program: msTimeSvc
 * File: msTimeSvc.c
 * Author: Blanton Radford
 * Created: December 05, 2014
 ********************************************************************
 * Implementation of program msTimeSvc
 ********************************************************************/

#ifdef _DEFAULT_INCLUDES
  #include <AsDefault.h>
#endif

_LOCAL BOOL running;    //  temporary
_LOCAL UDINT  run_ms;   //  temp

/*! \brief Init-SP for millisecond timer services
*   \pre   Place in TC#1 or first used TC
*/
void _INIT msTimeSvcInit(void)
{
  /* TODO: Add code here */
}

/*! \brief Cyclic task for millisecond timer services
*   \pre   Place in TC#1 or first used TC
*/
void _CYCLIC msTimeSvcCyclic(void)
{
 msTimer_typ * t=  &msTimer;

  t->clock_ms=  (UDINT)clock_ms();

  t->diff_ms= t->clock_ms - t->C1ms;

  t->C1ms=  t->clock_ms;

  // if(t->C1ms > 4294920000U)   t->C1ms=  0;      //  Keep absolute minute count accurate - WBR: check to see if this works
  if(t->C1ms > 4294920000U)   t->C1ms-= 4294920000U;      //  Keep absolute minute count accurate - WBR: check to see if this works
  //! \todo   inc t->C60sAbs?

  /// Calculate Other Counters
  t->C10ms=   t->C1ms / 10;
  t->C1s=     t->C1ms / 1000;
  t->C10s=    t->C1ms / 10000;
  t->C60s=    t->C1ms / 60000;

  // if(t->C60s > t->_old60s) t->C60sAbs++;
  if(t->C60s != t->_old60s) t->C60sAbs++;       //  should handle rollover
  t->_old60s=  t->C60s;

  ///  Calc pulse trains
  //  <boolean>=  ((t->C1ms % <period>) < <duration>);                          //  example - period and duration shall be in ms

  //  legacy
  t->F100ms=      ((t->C1ms %      100) <      50);
  t->F500ms=      ((t->C1ms %      500) <     250);
  t->F1s=         ((t->C1ms %     1000) <     500);
  t->F2s=         ((t->C1ms %     2000) <    1000);
  t->F10s=        ((t->C1ms %    10000) <    5000);

  //  new
  t->pulse01Hz100ms= ((t->C1ms % 1000) < 100);                                  //  WBR:  add these in the application as needed, or put frequently used ones here
  t->pulse1day100ms= ((t->C1ms % (24*3600*1000)) < 100);                        //  WBR:  comes on once per day for 100ms

  //! \todo   add configurable, periodic pulse(s), i.e. an (n)s pulse every (nn)min or (nn)day(s) or ???
  //! \todo   add hour meter(s)
  if(running)
  {
    run_ms+=  t->diff_ms;
  }
}
```

### Library Logical/Libraries/wbrServices/wbrListSvc (ANSIC)
Depends on: wbrsprintf, wbrMemSvc

### Program Logical/Libraries/wbrServices/wbrsprintf

#### cvtflasc.c
```c
/*
 *	cvtflasc - Convert floating-point to ASCII
 *
 *	arg		number to convert
 *	ndigits		number of digits to place in buffer
 *	decpt		place to return position of decimal point
 *	sign		place to return sign of number
 *	eflag		flag -- non-zero if `e' format should be used
 *	bufsize		size of `buf'
 *	buf		array in which to place result
 */

void __cvtflasc(double arg, int ndigits, int *decpt, int *sign, char eflag, int bufsize, char *buf)
	{
	int	exp10;		/* base 10 exponent of number		*/

	static const double roundvals[] =	/* values to add for rounding	*/
		{ 5.0e0, 5.0e-1, 5.0e-2, 5.0e-3, 5.0e-4, 5.0e-5,
		  5.0e-6, 5.0e-7, 5.0e-8, 5.0e-9, 5.0e-10, 5.0e-11,
		  5.0e-12, 5.0e-13, 5.0e-14, 5.0e-15, 5.0e-16, 5.0e-17,
		};
#define MAX (sizeof roundvals / sizeof *roundvals - 1)

	/* set sign
	 */
	if (arg < 0)
		{
		arg = -arg;
		*sign = 1;
		}
	else
		*sign = 0;

	/* Scale the number so it is in the range 1 to 10
	 */
	exp10 = 0;
	if (arg > 0)
		{
		while (arg >= 10)
			arg /= 10, ++exp10;
		while (arg < 1)
			arg *= 10, --exp10;
		}

	/* If `f' format, we want `ndigits' past the decimal point.
	 * If 'e' format we want ndigits + 1 digit before the decimal place.
	 */
	if (!eflag)
		ndigits += exp10 + 1;
	else
		++ndigits;

	/* Round the number to the specified number of digits
	 */
	arg += roundvals[ndigits > MAX ? MAX : ndigits];

	/* It might need more scaling after rounding
	 */
	if (arg >= 10)
		{
		arg = 1;
		++exp10;
		if (!eflag)
			++ndigits;
		}

	/* Set `decpt'
	 */
	*decpt = exp10 + 1;

	{
	register char *bufend = &buf[bufsize] - 1;
	register int c;
	register int i;

	for (i = 0 ; i < ndigits ; ++i)
		{
		if (buf >= bufend)
			break;
		if (i > 17)
			*buf++ = '0';
		else
			{
			c = (int)arg;
			*buf++ = '0' + c;
			arg = (arg - c) * 10;
			}
		}

	*buf = '\0';
	}

	}
```

### MTBasics.typ
```iecst
TYPE
	MTBasicsDT1InternalType : 	STRUCT  (*Internal variables of function block MTBasicsDT1.*)
		CycleTime : REAL; (*Task cycle time. Unit: [µs].*)
		ParametersValid : BOOL; (*Data for internal use.*)
		Gain : REAL; (*Data for internal use.*)
		TimeConstant : REAL; (*Data for internal use.*)
		Numerator : ARRAY[0..1]OF LREAL; (*Data for internal use.*)
		Denominator : ARRAY[0..1]OF LREAL; (*Data for internal use.*)
		BVector : ARRAY[0..1]OF LREAL; (*Data for internal use.*)
		AVector : ARRAY[0..1]OF LREAL; (*Data for internal use.*)
		XVector : ARRAY[0..1]OF LREAL; (*Data for internal use.*)
		PresetOK : BOOL; (*Data for internal use.*)
		PresetCoefficients : LREAL; (*Data for internal use.*)
		InOld : REAL; (*Data for internal use.*)
		UpdateOld : BOOL; (*Data for internal use.*)
		EnableOld : BOOL; (*Data for internal use.*)
		EnableDone : BOOL; (*Data for internal use.*)
		DisabledBusy : BOOL; (*Data for internal use.*)
		CounterOld : UDINT; (*Data for internal use.*)
		SysRefParaNew : BOOL; (*Data for internal use.*)
		SystemReference : MTTransferFcnType; (*Data for internal use.*)
	END_STRUCT;
	MTBasicsDT2InternalType : 	STRUCT  (*Internal variables of function block MTBasicsDT2.*)
		CycleTime : REAL; (*Task cycle time. Unit: [µs].*)
		ParametersValid : BOOL; (*Data for internal use.*)
		Gain : REAL; (*Data for internal use.*)
		TimeConstant1 : REAL; (*Data for internal use.*)
		TimeConstant2 : REAL; (*Data for internal use.*)
		Numerator : ARRAY[0..2]OF LREAL; (*Data for internal use.*)
		Denominator : ARRAY[0..2]OF LREAL; (*Data for internal use.*)
		BVector : ARRAY[0..2]OF LREAL; (*Data for internal use.*)
		AVector : ARRAY[0..2]OF LREAL; (*Data for internal use.*)
		XVector : ARRAY[0..1]OF LREAL; (*Data for internal use.*)
		PresetOK : BOOL; (*Data for internal use.*)
		PresetCoefficients : LREAL; (*Data for internal use.*)
		InOld : REAL; (*Data for internal use.*)
		UpdateOld : BOOL; (*Data for internal use.*)
		EnableOld : BOOL; (*Data for internal use.*)
		EnableDone : BOOL; (*Data for internal use.*)
		DisabledBusy : BOOL; (*Data for internal use.*)
		CounterOld : UDINT; (*Data for internal use.*)
		SysRefParaNew : BOOL; (*Data for internal use.*)
		SystemReference : MTTransferFcnType; (*Data for internal use.*)
	END_STRUCT;
	MTBasicsIntegratorInternalType : 	STRUCT  (*Internal variables of function block MTBasicsIntegrator.*)
		CycleTime : REAL; (*Task cycle time. Unit: [s].*)
		ParametersValid : BOOL; (*Data for internal use.*)
		Gain : REAL; (*Data for internal use.*)
		BVector : ARRAY[0..1]OF LREAL; (*Data for internal use.*)
		AVector : ARRAY[0..1]OF LREAL; (*Data for internal use.*)
		XVector : LREAL; (*Data for internal use.*)
		OutPresetValue : REAL; (*Data for internal use.*)
		SetOutOld : BOOL; (*Data for internal use.*)
		UpdateOld : BOOL; (*Data for internal use.*)
		EnableOld : BOOL; (*Data for internal use.*)
		EnableDone : BOOL; (*Data for internal use.*)
		DisabledBusy : BOOL; (*Data for internal use.*)
		CounterOld : UDINT; (*Data for internal use.*)
		SysRefParaNew : BOOL; (*Data for internal use.*)
		SystemReference : MTTransferFcnType; (*Data for internal use.*)
	END_STRUCT;
	MTBasicsLevelCtrlInternalType : 	STRUCT  (*Internal variables of function block MTBasicsLevelController.*)
		CycleTime : REAL; (*Task cycle time. Unit: [s].*)
		ParametersValid : BOOL; (*Data for internal use.*)
		Parameter : MTBasicsLevelCtrlParType; (*Data for internal use.*)
		State : USINT; (*Data for internal use.*)
		UpdateOld : BOOL; (*Data for internal use.*)
		EnableOld : BOOL; (*Data for internal use.*)
	END_STRUCT;
	MTBasicsLevelCtrlParType : 	STRUCT  (*Level controller parameters.*)
		OutputValue1 : REAL; (*1st Output value.*)
		OutputValue2 : REAL; (*2nd Output value.*)
		OutputValue3 : REAL; (*3rd Output value.*)
		ThresholdLevel1 : REAL; (*Threshold level from OutputValue2 to OutputValue1.*)
		ThresholdLevel2 : REAL; (*Threshold level from OutputValue1 to OutputValue2.*)
		ThresholdLevel3 : REAL; (*Threshold level from OutputValue3 to OutputValue2.*)
		ThresholdLevel4 : REAL; (*Threshold level from OutputValue2 to OutputValue3.*)
	END_STRUCT;
	MTBasicsLimiterInternalType : 	STRUCT  (*Internal variables of function block MTBasicsLimiter.*)
		CycleTime : REAL; (*Task cycle time. Unit: [s].*)
		ParametersValid : BOOL; (*Data for internal use.*)
		MaxOut : REAL; (*Data for internal use.*)
		MinOut : REAL; (*Data for internal use.*)
		MaxPosSlewRate : REAL; (*Data for internal use.*)
		MaxNegSlewRate : REAL; (*Data for internal use.*)
		Out : REAL; (*Data for internal use.*)
		OutOld : REAL; (*Data for internal use.*)
		UpperOutLimit : REAL; (*Data for internal use.*)
		LowerOutLimit : REAL; (*Data for internal use.*)
		SetOutOld : BOOL; (*Data for internal use.*)
		UpdateOld : BOOL; (*Data for internal use.*)
		EnableOld : BOOL; (*Data for internal use.*)
	END_STRUCT;
	MTBasicsOscTuningInternalType : 	STRUCT  (*Internal variables of function block MTBasicsOscillationTuning.*)
		CycleTime : REAL; (*Task cycle time. Unit: [s].*)
		ParametersValid : BOOL; (*Data for internal use.*)
		State : USINT; (*State of tuning.*)
		CriticalGain : REAL; (*Critical gain.*)
		OscillationPeriod : REAL; (*Period of oscillation.*)
		NumberOfOscillations : USINT; (*Number of osscilations.*)
		NumberOfPhases : USINT; (*Number of current tuning phase.*)
		MaxRelayOut : REAL; (*Lower limit for output during tuning.*)
		MinRelayOut : REAL; (*Upper limit for output during tuning.*)
		SetValue : REAL; (*Data for internal use.*)
		AverageOutValue : REAL; (*Data for internal use.*)
		MaxActValueTime : ARRAY[0..3]OF REAL; (*Data for internal use.*)
		MinActValueTime : ARRAY[0..3]OF REAL; (*Data for internal use.*)
		MaxActValue : ARRAY[0..3]OF REAL; (*Data for internal use.*)
		MinActValue : ARRAY[0..3]OF REAL; (*Data for internal use.*)
		TuningTime : REAL; (*Data for internal use.*)
		StartingActValue : REAL; (*Data for internal use.*)
		ControlError : REAL; (*Data for internal use.*)
		ActValueAverageAmplitude : REAL; (*Data for internal use.*)
		AverageActValue : REAL; (*Data for internal use.*)
		AverageMaxActValue : REAL; (*Data for internal use.*)
		AverageMinActValue : REAL; (*Data for internal use.*)
		AmplitudeRatio : REAL; (*Data for internal use.*)
		DeltaOut : REAL; (*Data for internal use.*)
		EffectiveDirection : SINT; (*Data for internal use.*)
		StartOld : BOOL; (*Data for internal use.*)
		MinOscillationAmplitude : REAL; (*Data for internal use.*)
		MinOut : REAL; (*Data for internal use.*)
		MaxOut : REAL; (*Data for internal use.*)
		TemporaryQuality : REAL; (*Data for internal use.*)
		TemporaryDerivativeTime : REAL; (*Data for internal use.*)
		TemporaryIntegrationTime : REAL; (*Data for internal use.*)
		TemporaryGain : REAL; (*Data for internal use.*)
		Update : BOOL; (*Data for internal use.*)
		UpdateOld : BOOL; (*Data for internal use.*)
		EnableOld : BOOL; (*Data for internal use.*)
		AverageOutValueSum : REAL; (*Data for internal use.*)
		AverageTime : LREAL; (*Data for internal use.*)
	END_STRUCT;
	MTBasicsPFMInternalType : 	STRUCT  (*Internal variables of function block MTBasicsPFM.*)
		CycleTime : REAL; (*Task cycle time. Unit: [s].*)
		ParametersValid : BOOL; (*Data for internal use.*)
		In : REAL; (*Data for internal use.*)
		PulseWidth : REAL; (*Data for internal use.*)
		MinPause : REAL; (*Data for internal use.*)
		Area : REAL; (*Data for internal use.*)
		AreaC : REAL; (*Data for internal use.*)
		OffTime : REAL; (*Data for internal use.*)
		OnTime : REAL; (*Data for internal use.*)
		Update : BOOL; (*Data for internal use.*)
		UpdateOld : BOOL; (*Data for internal use.*)
		EnableOld : BOOL; (*Data for internal use.*)
	END_STRUCT;
	MTBasicsPIDInternalType : 	STRUCT  (*Internal variables of function block MTBasicsPID.*)
		CycleTime : REAL; (*Task cycle time. Unit: [s].*)
		ParametersValid : BOOL; (*Data for internal use.*)
		PIDParameters : MTPIDParametersType; (*Data for internal use.*)
		MinOut : REAL; (*Data for internal use.*)
		MaxOut : REAL; (*Data for internal use.*)
		Invert : BOOL; (*Data for internal use.*)
		ControlError : REAL; (*Data for internal use.*)
		ControlErrorOld : REAL; (*Data for internal use.*)
		Out : REAL; (*Data for internal use.*)
		HoldIntegration : MTPIDIntegrationEnum; (*Data for internal use.*)
		IntegrationPartPresetValue : REAL; (*Data for internal use.*)
		SetIntegrationPart : BOOL; (*Data for internal use.*)
		SetIntegrationPartOld : BOOL; (*Data for internal use.*)
		EnableTrackingOld : BOOL; (*Data for internal use.*)
		PID_StatusID : DINT; (*Data for internal use.*)
		UpdateOld : BOOL; (*Data for internal use.*)
		EnableOld : BOOL; (*Data for internal use.*)
		EnableDone : BOOL; (*Data for internal use.*)
		DisabledBusy : BOOL; (*Data for internal use.*)
		CounterOld : UDINT; (*Data for internal use.*)
		SysRefParaNew : BOOL; (*Data for internal use.*)
		SystemReference : MTTransferFcnType; (*Data for internal use.*)
	END_STRUCT;
	MTBasicsPT1InternalType : 	STRUCT  (*Internal variables of function block MTBasicsPT1.*)
		CycleTime : REAL; (*Task cycle time. Unit: [s].*)
		ParametersValid : BOOL; (*Data for internal use.*)
		Gain : REAL; (*Data for internal use.*)
		TimeConstant : REAL; (*Data for internal use.*)
		Numerator : ARRAY[0..1]OF LREAL; (*Data for internal use.*)
		Denominator : ARRAY[0..1]OF LREAL; (*Data for internal use.*)
		BVector : ARRAY[0..1]OF LREAL; (*Data for internal use.*)
		AVector : ARRAY[0..1]OF LREAL; (*Data for internal use.*)
		XVector : ARRAY[0..1]OF LREAL; (*Data for internal use.*)
		OutPresetValue : REAL; (*Data for internal use.*)
		PresetCoefficients : LREAL; (*Data for internal use.*)
		PresetOK : BOOL; (*Data for internal use.*)
		SetOutOld : BOOL; (*Data for internal use.*)
		UpdateOld : BOOL; (*Data for internal use.*)
		EnableOld : BOOL; (*Data for internal use.*)
		EnableDone : BOOL; (*Data for internal use.*)
		DisabledBusy : BOOL; (*Data for internal use.*)
		CounterOld : UDINT; (*Data for internal use.*)
		SysRefParaNew : BOOL; (*Data for internal use.*)
		SystemReference : MTTransferFcnType; (*Data for internal use.*)
	END_STRUCT;
	MTBasicsPT2InternalType : 	STRUCT  (*Internal variables of function block MTBasicsPT2.*)
		CycleTime : REAL; (*Task cycle time. Unit: [µs].*)
		ParametersValid : BOOL; (*Data for internal use.*)
		Gain : REAL; (*Data for internal use.*)
		TimeConstant1 : REAL; (*Data for internal use.*)
		TimeConstant2 : REAL; (*Data for internal use.*)
		Numerator : ARRAY[0..2]OF LREAL; (*Data for internal use.*)
		Denominator : ARRAY[0..2]OF LREAL; (*Data for internal use.*)
		BVector : ARRAY[0..2]OF LREAL; (*Data for internal use.*)
		AVector : ARRAY[0..2]OF LREAL; (*Data for internal use.*)
		XVector : ARRAY[0..1]OF LREAL; (*Data for internal use.*)
		OutPresetValue : REAL; (*Data for internal use.*)
		PresetCoefficients : LREAL; (*Data for internal use.*)
		PresetOK : BOOL; (*Data for internal use.*)
		SetOutOld : BOOL; (*Data for internal use.*)
		UpdateOld : BOOL; (*Data for internal use.*)
		EnableOld : BOOL; (*Data for internal use.*)
		EnableDone : BOOL; (*Data for internal use.*)
		DisabledBusy : BOOL; (*Data for internal use.*)
		CounterOld : UDINT; (*Data for internal use.*)
		SysRefParaNew : BOOL; (*Data for internal use.*)
		SystemReference : MTTransferFcnType; (*Data for internal use.*)
	END_STRUCT;
	MTBasicsPWMInternalType : 	STRUCT  (*Internal variables of function block MTBasicsPWM.*)
		CycleTime : REAL; (*Task cycle time. Unit: [s].*)
		ParametersValid : BOOL; (*Data for internal use.*)
		Mode : MTBasicsPWMModeEnum; (*Data for internal use.*)
		MinPulseWidth : REAL; (*Data for internal use.*)
		Period : REAL; (*Data for internal use.*)
		In : REAL; (*Data for internal use.*)
		OnTime : REAL; (*Data for internal use.*)
		OffTime : REAL; (*Data for internal use.*)
		PeriodCounter : REAL; (*Data for internal use.*)
		OnTimeCounter : REAL; (*Data for internal use.*)
		UpdateOld : BOOL; (*Data for internal use.*)
		EnableOld : BOOL; (*Data for internal use.*)
	END_STRUCT;
	MTBasicsPWMModeEnum :
		( (*Pulse mode.*)
		mtBASICS_PULSE_BEGINNING := 0, (*Pulse at the beginning of a period.*)
		mtBASICS_PULSE_MIDDLE := 1 (*Pulse in the middle of a period.*)
		);
	MTBasicsPWMScheduleBufferPtrType : 	STRUCT  (*Buffer pointers of the PWMSchedule.*)
		In : REAL; (*Data for internal use.*)
		OnTime1 : REAL; (*Data for internal use.*)
		OnTime2 : REAL; (*Data for internal use.*)
		OffTime1 : REAL; (*Data for internal use.*)
		OffTime2 : REAL; (*Data for internal use.*)
		OnTimeCounter : REAL; (*Data for internal use.*)
	END_STRUCT;
	MTBasicsPWMScheduleBufferType : 	STRUCT  (*Buffer parameters of the PWMSchedule.*)
		ActIndex : UINT; (*Data for internal use.*)
		ActBufferElements : UINT; (*Data for internal use.*)
		OldBufferElements : {REDUND_UNREPLICABLE} UINT; (*Data for internal use.*)
		PointerTimes : REFERENCE TO MTBasicsPWMScheduleBufferPtrType; (*Data for internal use.*)
		PointerOut : REFERENCE TO BOOL; (*Data for internal use.*)
	END_STRUCT;
	MTBasicsPWMScheduleInternalType : 	STRUCT  (*Internal variables of function block MTBasicsPWM.*)
		CycleTime : REAL; (*Task cycle time. Unit: [s].*)
		ParametersValid : BOOL; (*Data for internal use.*)
		NumberOfInputs : UINT; (*Data for internal use.*)
		Mode : MTBasicsPWMScheduleModeEnum; (*Data for internal use.*)
		MinPulseWidth : REAL; (*Data for internal use.*)
		MinPause : REAL; (*Data for internal use.*)
		Period : REAL; (*Data for internal use.*)
		FreeDutyCycle : REAL; (*Data for internal use.*)
		PeriodCounter : REAL; (*Data for internal use.*)
		Buffer : MTBasicsPWMScheduleBufferType; (*Data for internal use.*)
		UpdateOld : BOOL; (*Data for internal use.*)
		EnableOld : {REDUND_UNREPLICABLE} BOOL; (*Data for internal use.*)
		InhibitUpdate : BOOL; (*Data for internal use.*)
		Update : BOOL; (*Data for internal use.*)
		StatusIDUpdate : DINT; (*Data for internal use.*)
	END_STRUCT;
	MTBasicsPWMScheduleModeEnum :
		( (*Schedule mode.*)
		mtBASICS_SHIFT_PULSE := 0, (*Shift the puls.*)
		mtBASICS_SPLIT_PULSE := 1 (*Split the puls.*)
		);
	MTBasicsStepTuningBufElemType : 	STRUCT  (*Buffer element of MTBasicsStepTuning.*)
		TimeIndex : UDINT; (*Data for internal use.*)
		In : LREAL; (*Data for internal use.*)
		IntIn : LREAL; (*Data for internal use.*)
		IntTimeIn : LREAL; (*Data for internal use.*)
		IntTime2In : LREAL; (*Data for internal use.*)
		Int2In : LREAL; (*Data for internal use.*)
		Int3In : LREAL; (*Data for internal use.*)
		TSum : LREAL; (*Data for internal use.*)
		dTSum : LREAL; (*Data for internal use.*)
		d2TSum : LREAL; (*Data for internal use.*)
		dyACD : LREAL; (*Data for internal use.*)
		d2yACD : LREAL; (*Data for internal use.*)
		d3yACD : LREAL; (*Data for internal use.*)
		DiffIn : LREAL; (*Data for internal use.*)
		Diff2In : LREAL; (*Data for internal use.*)
	END_STRUCT;
	MTBasicsStepTuningInternalType : 	STRUCT  (*Internal variables of function block MTBasicsStepTuning.*)
		CycleTime : REAL; (*Task cycle time. Unit: [s].*)
		ParametersValid : BOOL; (*Data for internal use.*)
		MinActValue : REAL; (*Data for internal use.*)
		MaxActValue : REAL; (*Data for internal use.*)
		MaxTuningTime : REAL; (*Data for internal use.*)
		StepHeight : REAL; (*Data for internal use.*)
		State : MTBasicsStepTuningStateEnum; (*Data for internal use.*)
		TuningTime : REAL; (*Data for internal use.*)
		Area : REAL; (*Data for internal use.*)
		StartActValue : REAL; (*Data for internal use.*)
		SumTime : REAL; (*Data for internal use.*)
		PlantGain : REAL; (*Data for internal use.*)
		LQError : REAL; (*Data for internal use.*)
		LQOutput : ARRAY[0..1]OF REAL; (*Data for internal use.*)
		LQParameterVector : ARRAY[0..2]OF REAL; (*Data for internal use.*)
		ActValueOld : REAL; (*Data for internal use.*)
		SystemSettlingTime : REAL; (*Data for internal use.*)
		SettlingIndex : UINT; (*Data for internal use.*)
		NumberOfSettlingValues : UINT; (*Data for internal use.*)
		NoiseDeadBand : REAL; (*Data for internal use.*)
		StartOld : BOOL; (*Data for internal use.*)
		UpdateOld : BOOL; (*Data for internal use.*)
		EnableOld : BOOL; (*Data for internal use.*)
		Slope : REAL; (*Data for internal use.*)
	END_STRUCT;
	MTBasicsStepTuningStateEnum :
		( (*Tuning state.*)
		mtBASICS_STATE_READY := 1, (*The function block waits for a rising edge of Start.*)
		mtBASICS_STATE_SETTLING := 2, (*It is checked, if the system is in an idle state.*)
		mtBASICS_STATE_STEP := 3, (*The output Out is set to the value StepHeight.*)
		mtBASICS_STATE_CALCULATE_PID := 4 (*PID parameters are calculated.*)
		);
	MTBasicsTimeDelayFcnParaType : 	STRUCT  (*Internal variables for time delay function parameters.*)
		DelayCounter : UDINT; (*Data for internal use.*)
		ActBufferIndex : UDINT; (*Data for internal use.*)
		ActBufferElements : UDINT; (*Data for internal use.*)
		OldBufferElements : UDINT; (*Data for internal use.*)
		DelayTimeAct : REAL; (*Data for internal use.*)
		BufferPointer : REFERENCE TO REAL; (*Data for internal use.*)
	END_STRUCT;
	MTBasicsTimeDelayInternalType : 	STRUCT  (*Internal variables of function block MTBasicsTimeDelay.*)
		CycleTime : REAL; (*Task cycle time. Unit: [s].*)
		DelayTime : REAL; (*Data for internal use.*)
		ParametersValid : BOOL; (*Data for internal use.*)
		InitialValue : REAL; (*Data for internal use.*)
		EnableOld : BOOL; (*Data for internal use.*)
		TimeDelayFcnPara : {REDUND_UNREPLICABLE} MTBasicsTimeDelayFcnParaType; (*Data for internal use.*)
	END_STRUCT;
END_TYPE
```

### MTBasics.var
```iecst
(*Error*)
VAR CONSTANT
	mtBCD_ERR_TIME_CONSTANT1_INVALID : DINT := -1058012139; (*Chosen first time constant is invalid.*)
	mtBCD_ERR_TIME_CONSTANT2_INVALID : DINT := -1058012138; (*Chosen second time constant is invalid.*)
	mtBCD_ERR_THRESHOLD_NOT_DEFINED : DINT := -1058012137; (*Chosen values for the threshold levels are invalid.*)
	mtBCD_ERR_THRESHOLD_INVALID : DINT := -1058012136; (*One of the values for the threshold levels is invalid.*)
	mtBCD_ERR_OUT_VALUE_NOT_DEFINED : DINT := -1058012135; (*Chosen output values are invalid.*)
	mtBCD_ERR_OUTPUT_LIMIT_INVALID : DINT := -1058012134; (*Chosen limitations for output are invalid.*)
	mtBCD_ERR_MAX_POS_SLEW_RATE_NEG : DINT := -1058012133; (*Chosen slew rate for positive direction is invalid.*)
	mtBCD_ERR_MAX_NEG_SLEW_RATE_NEG : DINT := -1058012132; (*Chosen slew rate for negative direction is invalid.*)
	mtBCD_ERR_PULSE_WIDTH_LOW : DINT := -1058012131; (*Chosen pulse width is too low.*)
	mtBCD_ERR_MIN_PAUSE_LOW : DINT := -1058012130; (*The selected minimum pause duration is too low.*)
	mtBCD_ERR_MIN_PULSE_HIGH : DINT := -1058012124; (*The selected minimum pulse duration is too high.*)
	mtBCD_ERR_MIN_PULSE_LOW : DINT := -1058012123; (*The selected minimum pulse duration is too low.*)
	mtBCD_ERR_PERIOD_LOW : DINT := -1058012122; (*The selected period duration is too low.*)
	mtBCD_ERR_NUMBER_OF_INPUTS : DINT := -1058012121; (*The selected number of inputs is invalid.*)
	mtBCD_ERR_SAMPLING_INVALID : DINT := -1058012118; (*The period of the generated oscillation is invalid. *)
	mtBCD_ERR_SETTLING_TIME_INVALID : DINT := -1058012117; (*Chosen duration, in which the settling of the system is detected, is invalid.*)
	mtBCD_ERR_TUNING_TIME_INVALID : DINT := -1058012116; (*Chosen maximum tuning time is invalid.*)
	mtBCD_ERR_ACT_VALUE_NOT_STABLE : DINT := -1058012115; (*The system is not in a settled operating point.*)
	mtBCD_ERR_RANGE_INVALID : DINT := -1058012114; (*Chosen limitations for the input are invalid.*)
	mtBCD_ERR_TUNING_INVALID : DINT := -1058012113; (*Tuning was not successful.*)
	mtBCD_ERR_MIN_PAUSE_HIGH : DINT := -1058012112; (*The selected minimum pause duration is too high.*)
	mtBCD_ERR_MODE_INVALID : DINT := -1058012111; (*The selected mode is invalid.*)
	mtBCD_ERR_NULL_PTR : DINT := -1058012110; (*Null pointer passed to the input.*)
END_VAR
(*Warning*)
VAR CONSTANT
	mtBCD_WRN_TIME_CONSTANT1_INVALID : DINT := -2131753963; (*Chosen first time constant is invalid.*)
	mtBCD_WRN_TIME_CONSTANT2_INVALID : DINT := -2131753962; (*Chosen second time constant is invalid.*)
	mtBCD_WRN_THRESHOLD_NOT_DEFINED : DINT := -2131753961; (*Chosen values for the threshold levels are invalid.*)
	mtBCD_WRN_THRESHOLD_INVALID : DINT := -2131753960; (*One of the values for the threshold levels is invalid.*)
	mtBCD_WRN_OUT_VALUE_NOT_DEFINED : DINT := -2131753959; (*Chosen output values are invalid.*)
	mtBCD_WRN_OUTPUT_LIMIT_INVALID : DINT := -2131753958; (*Chosen limitations for output are invalid.*)
	mtBCD_WRN_MAX_POS_SLEW_RATE_NEG : DINT := -2131753957; (*Chosen slew rate for positive direction is invalid.*)
	mtBCD_WRN_MAX_NEG_SLEW_RATE_NEG : DINT := -2131753956; (*Chosen slew rate for negative direction is invalid.*)
	mtBCD_WRN_PULSE_WIDTH_LOW : DINT := -2131753955; (*Chosen pulse width is too low.*)
	mtBCD_WRN_MIN_PAUSE_LOW : DINT := -2131753954; (*The selected minimum pause duration is too low.*)
	mtBCD_WRN_GAIN_ZERO : DINT := -2131753953; (*Chosen gain is zero.*)
	mtBCD_WRN_FILTER_TIME_LOW : DINT := -2131753948; (*Chosen filter time is invalid.*)
	mtBCD_WRN_MIN_PULSE_HIGH : DINT := -2131753946; (*The selected minimum pulse duration is too high.*)
	mtBCD_WRN_MIN_PULSE_LOW : DINT := -2131753945; (*The selected minimum pulse duration is too low.*)
	mtBCD_WRN_PERIOD_LOW : DINT := -2131753944; (*The selected period duration is too low.*)
	mtBCD_WRN_SETTLING_TIME_INVALID : DINT := -2131753941; (*Chosen duration, in which the settling of the system is detected, is invalid.*)
	mtBCD_WRN_TUNING_TIME_INVALID : DINT := -2131753940; (*Chosen maximum tuning time is invalid.*)
	mtBCD_WRN_STEP_HEIGHT_INVALID : DINT := -2131753939; (*Chosen step height is zero.*)
	mtBCD_WRN_RANGE_INVALID : DINT := -2131753938; (*Chosen limitations for the input are invalid.*)
	mtBCD_WRN_MIN_PAUSE_HIGH : DINT := -2131753937; (*The selected minimum pause duration is too high.*)
	mtBCD_WRN_MODE_INVALID : DINT := -2131753936; (*The selected mode is invalid.*)
END_VAR
(*Information*)
VAR CONSTANT
	mtBCD_INF_TIME_CONSTANT1_ZERO : DINT := 1089471509; (*Operating as P element or PT1 / DT1 element since TimeConstant1 = 0.*)
	mtBCD_INF_TIME_CONSTANT2_ZERO : DINT := 1089471510; (*Operating as P element or PT1 / DT1 element since TimeConstant2 = 0.*)
	mtBCD_INF_TUNING_ABORTED_BY_USER : DINT := 1089471511; (*Tuning aborted by user.*)
END_VAR
```

### MTFilter.typ
```iecst
TYPE
	MTFilterMovingAvgInternalType : 	STRUCT  (*Internal variables of function block MTFilterMovingAverage.*)
		Ts : REAL; (*Data for internal use.*)
		ParameterValid : BOOL; (*Data for internal use.*)
		NumOfElmements : UINT; (*Number of elements of calculating output.*)
		Sum : LREAL; (*Data for internal use.*)
		pBuffer : {REDUND_UNREPLICABLE} UDINT; (*Data for internal use.*)
		CntAct : UINT; (*Data for internal use.*)
		CntOld : UINT; (*Data for internal use.*)
		WindowLength : UINT; (*Data for internal use.*)
		BufferLength : UINT; (*Length of window.*)
		BufferFull : BOOL; (*Data for internal use.*)
		MemAllocated : BOOL; (*Data for internal use.*)
		Update : BOOL; (*Data for internal use.*)
		UpdateOld : BOOL; (*Data for internal use.*)
		EnableOld : BOOL; (*Data for internal use.*)
		statusTMP : UINT; (*Data for internal use.*)
	END_STRUCT;
	MTFilterTypeEnum :
		( (*Filtertype.*)
		mtFILTER_BESSEL := 0, (*Bessel Filter.*)
		mtFILTER_BUTTERWORTH := 1 (*Butterworth Filter.*)
		);
	MTFilterLowPassInternalType : 	STRUCT  (*Internal variables of function block MTFilterLowPass.*)
		Ts : REAL; (*Task cycle time. Unit: [s].*)
		SamplingFrequency : LREAL; (*Sampling frequency. Unit: [Hz].*)
		ParameterValid : BOOL; (*Data for internal use.*)
		AngularFrequency : LREAL; (*Data for internal use.*)
		Num : ARRAY[0..5]OF LREAL; (*Data for internal use.*)
		Den : ARRAY[0..5]OF LREAL; (*Data for internal use.*)
		BVector : ARRAY[0..5]OF LREAL; (*Data for internal use.*)
		AVector : ARRAY[0..5]OF LREAL; (*Data for internal use.*)
		XVector : ARRAY[0..4]OF LREAL; (*Data for internal use.*)
		TypeOld : USINT; (*Data for internal use.*)
		OrderOld : USINT; (*Data for internal use.*)
		CutOffFrequencyOld : REAL; (*Data for internal use.*)
		UpdateOld : BOOL; (*Data for internal use.*)
		EnableOld : BOOL; (*Data for internal use.*)
		EnableDone : BOOL; (*Data for internal use.*)
		DisabledBusy : BOOL; (*Data for internal use.*)
		CounterOld : UDINT; (*Data for internal use.*)
		SysRefParaNew : BOOL; (*Data for internal use.*)
		SystemReference : MTTransferFcnType; (*Data for internal use.*)
	END_STRUCT;
	MTFilterHighPassInternalType : 	STRUCT  (*Internal variables of function block MTFilterHighPass.*)
		Ts : REAL; (*Task cycle time. Unit: [s].*)
		SamplingFrequency : LREAL; (*Sampling frequency. Unit: [Hz].*)
		ParameterValid : BOOL; (*Data for internal use.*)
		AngularFrequency : LREAL; (*Frequency in radians*)
		Num : ARRAY[0..5]OF LREAL; (*Data for internal use.*)
		Den : ARRAY[0..5]OF LREAL; (*Data for internal use.*)
		BVector : ARRAY[0..5]OF LREAL; (*Data for internal use.*)
		AVector : ARRAY[0..5]OF LREAL; (*Data for internal use.*)
		XVector : ARRAY[0..4]OF LREAL; (*Data for internal use.*)
		TypeOld : USINT; (*Data for internal use.*)
		OrderOld : USINT; (*Data for internal use.*)
		CutOffFrequencyOld : REAL; (*Data for internal use.*)
		UpdateOld : BOOL; (*Data for internal use.*)
		EnableOld : BOOL; (*Data for internal use.*)
		EnableDone : BOOL; (*Data for internal use.*)
		DisabledBusy : BOOL; (*Data for internal use.*)
		CounterOld : UDINT; (*Data for internal use.*)
		SysRefParaNew : BOOL; (*Data for internal use.*)
		SystemReference : MTTransferFcnType; (*Data for internal use.*)
	END_STRUCT;
	MTFilterBandPassInternalType : 	STRUCT  (*Internal variables of function block MTFilterBandPass.*)
		Ts : REAL; (*Task cycle time. Unit: [s].*)
		SamplingFrequency : LREAL; (*Sampling frequency. Unit: [Hz].*)
		ParameterValid : BOOL; (*Data for internal use.*)
		AngularFrequency : LREAL; (*Frequency in radians*)
		BandwidthRad : LREAL; (*Frequency in radians*)
		Num : ARRAY[0..5]OF LREAL; (*Data for internal use.*)
		Den : ARRAY[0..5]OF LREAL; (*Data for internal use.*)
		BVector : ARRAY[0..5]OF LREAL; (*Data for internal use.*)
		AVector : ARRAY[0..5]OF LREAL; (*Data for internal use.*)
		XVector : ARRAY[0..4]OF LREAL; (*Data for internal use.*)
		TypeOld : USINT; (*Data for internal use.*)
		OrderOld : USINT; (*Data for internal use.*)
		CenterFrequencyOld : REAL; (*Data for internal use.*)
		BandwidthOld : REAL; (*Data for internal use.*)
		UpdateOld : BOOL; (*Data for internal use.*)
		EnableOld : BOOL; (*Data for internal use.*)
		EnableDone : BOOL; (*Data for internal use.*)
		DisabledBusy : BOOL; (*Data for internal use.*)
		CounterOld : UDINT; (*Data for internal use.*)
		SysRefParaNew : BOOL; (*Data for internal use.*)
		SystemReference : MTTransferFcnType; (*Data for internal use.*)
	END_STRUCT;
	MTFilterBandStopInternalType : 	STRUCT  (*Internal variables of function block MTFilterBandStop.*)
		Ts : REAL; (*Task cycle time. Unit: [s].*)
		SamplingFrequency : LREAL; (*Sampling frequency. Unit: [Hz].*)
		ParameterValid : BOOL; (*Data for internal use.*)
		AngularFrequency : LREAL; (*Data for internal use.*)
		BandwidthRad : LREAL; (*Frequency in radians*)
		Num : ARRAY[0..5]OF LREAL; (*Data for internal use.*)
		Den : ARRAY[0..5]OF LREAL; (*Data for internal use.*)
		BVector : ARRAY[0..5]OF LREAL; (*Data for internal use.*)
		AVector : ARRAY[0..5]OF LREAL; (*Data for internal use.*)
		XVector : ARRAY[0..4]OF LREAL; (*Data for internal use.*)
		TypeOld : USINT; (*Data for internal use.*)
		OrderOld : USINT; (*Data for internal use.*)
		CenterFrequencyOld : REAL; (*Data for internal use.*)
		BandwidthOld : REAL; (*Data for internal use.*)
		UpdateOld : BOOL; (*Data for internal use.*)
		EnableOld : BOOL; (*Data for internal use.*)
		EnableDone : BOOL; (*Data for internal use.*)
		DisabledBusy : BOOL; (*Data for internal use.*)
		CounterOld : UDINT; (*Data for internal use.*)
		SysRefParaNew : BOOL; (*Data for internal use.*)
		SystemReference : MTTransferFcnType; (*Data for internal use.*)
	END_STRUCT;
	MTFilterNotchInternalType : 	STRUCT  (*Internal variables of function block MTFilterNotch.*)
		Ts : REAL; (*Task cycle time. Unit: [s].*)
		SamplingFrequency : LREAL; (*Sampling frequency. Unit: [Hz].*)
		ParametersValid : BOOL; (*Data for internal use.*)
		UpperFrequency : REAL; (*Data for internal use.*)
		LowerFrequency : REAL; (*Data for internal use.*)
		BandwidthAct : REAL; (*Data for internal use.*)
		DampingConstant : REAL; (*Data for internal use.*)
		FilterTimeConstant : REAL; (*Data for internal use.*)
		Num : ARRAY[0..2]OF LREAL; (*Data for internal use.*)
		Den : ARRAY[0..2]OF LREAL; (*Data for internal use.*)
		BVector : ARRAY[0..2]OF LREAL; (*Data for internal use.*)
		AVector : ARRAY[0..2]OF LREAL; (*Data for internal use.*)
		XVector : ARRAY[0..1]OF LREAL; (*Data for internal use.*)
		TypeOld : USINT; (*Data for internal use.*)
		OrderOld : USINT; (*Data for internal use.*)
		CutOffFrequencyOld : REAL; (*Data for internal use.*)
		UpdateOld : BOOL; (*Data for internal use.*)
		EnableOld : BOOL; (*Data for internal use.*)
		EnableDone : BOOL; (*Data for internal use.*)
		DisabledBusy : BOOL; (*Data for internal use.*)
		SysRefParaNew : BOOL; (*Data for internal use.*)
		CounterOld : UDINT; (*Data for internal use.*)
		SystemReference : MTTransferFcnType; (*Data for internal use.*)
	END_STRUCT;
	MTFilterBiQuadInternalType : 	STRUCT  (*Internal variables of function block MTFilterBiQuad.*)
		Ts : REAL; (*Task cycle time. Unit: [s].*)
		SamplingFrequency : LREAL; (*Sampling frequency. Unit: [Hz]*)
		ParameterValid : BOOL; (*Data for internal use.*)
		Num : ARRAY[0..2]OF LREAL; (*Data for internal use.*)
		Den : ARRAY[0..2]OF LREAL; (*Data for internal use.*)
		BVector : ARRAY[0..2]OF LREAL; (*Data for internal use.*)
		AVector : ARRAY[0..2]OF LREAL; (*Data for internal use.*)
		XVector : ARRAY[0..1]OF LREAL; (*Data for internal use.*)
		FrequencyNumeratorOld : REAL; (*Data for internal use.*)
		DampingRatioNumeratorOld : REAL; (*Data for internal use.*)
		FrequencyDenominatorOld : REAL; (*Data for internal use.*)
		DampingRatioDenominatorOld : REAL; (*Data for internal use.*)
		FrequencyNumeratorRad : LREAL; (*Data for internal use.*)
		FrequencyDenominatorRad : LREAL; (*Data for internal use.*)
		UpdateOld : BOOL; (*Data for internal use.*)
		EnableOld : BOOL; (*Data for internal use.*)
		EnableDone : BOOL; (*Data for internal use.*)
		DisabledBusy : BOOL; (*Data for internal use.*)
		SysRefParaNew : BOOL; (*Data for internal use.*)
		CounterOld : UDINT; (*Data for internal use.*)
		SystemReference : MTTransferFcnType; (*Data for internal use.*)
	END_STRUCT;
END_TYPE
```

### Program Logical/Application/Creaser (IEC)

#### Main.st - Init, cyclic, exit code
```iecst
PROGRAM _INIT

	Action_Init_Infeed_Axis; //Set pointer values/initialize servo drive FBK MpAxisBasic instance

	MachineState := MACHINE_STATE_INIT;

	Pulse_Slow.TimeOn := DEFINE_SLOW_PULSE_PERIOD;
	Pulse_Slow.TimeOff := DEFINE_SLOW_PULSE_PERIOD;

	Pulse_Fast.TimeOn := DEFINE_FAST_PULSE_PERIOD;
	Pulse_Fast.TimeOff := DEFINE_FAST_PULSE_PERIOD;

	StdDevCalc.Enable := TRUE;

END_PROGRAM

PROGRAM _CYCLIC

	IF gStatistics.Reset THEN //Reset all statistics
		brsmemset(ADR(gStatistics), 0, SIZEOF(Global_Statistics_typ)); //Kind of a weird way to do this- essentially just writes 0's to the entirety of the memory the structure occupies (thus "zeroing-out" the counters)
		StdDevCalc.Enable := TRUE;
		StdDevCalc.Reset := FALSE;
		StdDevCalc();
		StdDevCalc.Reset := TRUE;
		StdDevCalc();
		StdDevCalc.Reset := FALSE;
	END_IF;

	Action_Eval_ErrorState_Statuses; //Evaluate the conditions that put machine into ERR state

	//Eval conditions that would send the machine into ERR state if the machine isn't already in ERR or INIT state->

	IF EDGEPOS(IO.iSafeMachineState) OR iMachineErrorReset THEN
		ProcessState := PRCS_STATE_INIT;
		gAlarmResetRequested := TRUE;
		//		gStatistics.Reset := TRUE;
		MachineState := MACHINE_STATE_INIT;
	END_IF;

	IF EDGEPOS(MachineState = MACHINE_STATE_ERROR) THEN
		AxisControl.MoveVelocity := FALSE;
		AxisControl.MoveAbsolute := FALSE;
		AxisControl.MoveAdditive := FALSE;
		AxisControl.Stop := TRUE;
		AxisControl();
	END_IF;

	BoardEjectUIButton_Hide := BOOL_TO_USINT(NOT ((MachineState = MACHINE_STATE_IDLE OR MachineState = MACHINE_STATE_MANUAL_EJECT) AND IO.iFiberOpticSensor));

	StartUIButton_Hide := NOT (MachineState = MACHINE_STATE_IDLE);
	StopUIButton_Hide := NOT (MachineState = MACHINE_STATE_RUNNING);

	Action_Tally_Board_L;

	CASE MachineState OF
		MACHINE_STATE_INIT:
			IO.oBoardFeedingLight := FALSE;
			IO.oUIIndicatorLight := FALSE;
			AxisControl.Power := FALSE;

			MachineState := MACHINE_STATE_HARDWARE_INIT;

		MACHINE_STATE_HARDWARE_INIT:
			IO.oBoardFeedingLight := FALSE;
			IO.oUIIndicatorLight := FALSE;

			IF AxisControl.Info.ReadyToPowerOn THEN
				AxisControl.Power := TRUE;
				MachineState := MACHINE_STATE_AXIS_POWER;
			END_IF;

		MACHINE_STATE_AXIS_POWER:
			IO.oBoardFeedingLight := FALSE;
			IO.oUIIndicatorLight := FALSE;

			IF AxisControl.PowerOn THEN
				Action_Stop_Feeder;
				MachineState := MACHINE_STATE_IDLE;
			END_IF;

		MACHINE_STATE_IDLE:
			IO.oBoardFeedingLight := FALSE;
			IO.oUIIndicatorLight := Pulse_Slow.bFlashOut;

			IF EDGEPOS(iManualBoardEject) THEN

				AxisControl.MoveVelocity := FALSE;
				AxisControl.MoveAbsolute := FALSE;
				AxisControl.MoveAdditive := FALSE;
				AxisControl.Stop := FALSE;
				AxisControl();

				AxisPar.Velocity := gRecCfg.active.Rec.FeedVelocity;
				AxisPar.Acceleration := gRecCfg.active.Cfg.Creaser.FeedAxisAccel;
				AxisPar.Deceleration := gRecCfg.active.Cfg.Creaser.FeedAxisDecel;

				AxisControl.MoveVelocity := TRUE;
				AxisControl();

				MachineState := MACHINE_STATE_MANUAL_EJECT;
			END_IF;

			IF EDGEPOS(iStartCommand) THEN
				IF IO.iFiberOpticSensor THEN
					gAlarms.Fiber_Optic_Blocked_RunCmd := TRUE;
					MachineState := MACHINE_STATE_ERROR;
				ELSIF NOT IO.iCreaserShaftSensor THEN
					gAlarms.Manual_Home_Creaser_Blade := TRUE;
					MachineState := MACHINE_STATE_ERROR;
				ELSE
					//					setflagCreaserIndexCommand := TRUE;
					iSoftStopCommand := FALSE;
					Action_Start_Feeder;
					ProcessState := PRCS_STATE_INIT;
					MachineState := MACHINE_STATE_RUNNING;
				END_IF;
			END_IF;

		MACHINE_STATE_MANUAL_EJECT:
			IO.oBoardFeedingLight := TRUE;
			IO.oUIIndicatorLight := Pulse_Slow.bFlashOut;

			IF (NOT IO.iFiberOpticSensor AND IO_LastCycle.iFiberOpticSensor) OR NOT iManualBoardEject THEN
				Action_Stop_Feeder;
				MachineState := MACHINE_STATE_IDLE;
			END_IF;

		MACHINE_STATE_RUNNING:
			IO.oUIIndicatorLight := TRUE;

			Action_Manage_Update_Total_Runtime;

			IF iSoftStopCommand THEN

				IF NOT (ProcessState = PRCS_STATE_SOFT_STOP) THEN
					Action_Stop_Feeder;
				END_IF;

				ProcessState := PRCS_STATE_SOFT_STOP;
			END_IF;

			Action_CreaserProcess_SM; //Crease motor <-> movement cycle <-> FiOS state machine

		MACHINE_STATE_ERROR: //ERROR state.  Note that this state is exited via the logic ABOVE the state machine.
			IO.oBoardFeedingLight := FALSE;
			IO.oUIIndicatorLight := Pulse_Fast.bFlashOut AND Pulse_Slow.bFlashOut;

			Current_Crease_Section_Length := 0;

			ProcessState := PRCS_STATE_INIT;

	END_CASE;

	Pulse_Slow;
	Pulse_Fast;

	Action_Creaser_Idx; //Reads/sets flag variables indicating current state of the creasing motor
	Action_AxisControl_Mgmt; //Calls Infeed Axis Control FBK, sets/resets drive errors

	IO_LastCycle := IO; //Latch previous cycle IO values (since EDGEPOS() has some weird caveats)
END_PROGRAM

PROGRAM _EXIT
	(* Insert code here *)

END_PROGRAM
```

#### Variables.var - Local variables
```iecst
VAR
	Timer_Sim_CreaserIdx : TON;
	Timer_Creaser_Idx_Edge : TON;
	Timer_Total_Runtime : TON;
	tmp_bool : BOOL;
END_VAR
(*Insert your comment here.*)
VAR
	setFlagTravelEdgeOffset : BOOL;
	setFlagCreaserIdxFinished : BOOL;
	setflagCreaserIndexCommand : BOOL;
	setFlagCreaserWaitEdge : BOOL;
END_VAR
(*Insert your comment here.*)
VAR
	flagBoardLengthCfgErr : BOOL;
	length_calculated_total : REAL;
END_VAR
VAR CONSTANT
	DEFINE_SLOW_PULSE_PERIOD : TIME := T#1s;
	DEFINE_FAST_PULSE_PERIOD : TIME := T#125ms;
END_VAR
VAR
	Pulse_Slow : PulseTrain;
	Pulse_Fast : PulseTrain;
	ii_crease_count : UDINT;
END_VAR
```

#### Action_Manage_Update_Total_Runtime.st - Manage the total runtime counter and its breakdown into HH:MM:SS
```iecst
ACTION Action_Manage_Update_Total_Runtime:

	IF bgTimerIsTimeOut(Timer_Total_Runtime) THEN
		gStatistics.total_runtime := gStatistics.total_runtime + 1;
		bgTimerStart(Timer_Total_Runtime, 1000);

		gStatistics.runtime_h := gStatistics.total_runtime / 3600;
		gStatistics.runtime_m := gStatistics.total_runtime 	MOD 3600;
		gStatistics.runtime_s := gStatistics.total_runtime MOD 60;
	END_IF;

	bgTimerCyclic(Timer_Total_Runtime);

END_ACTION
```

#### Action_Start_Feeder.st
```iecst
ACTION Action_Start_Feeder:
	AxisPar.Velocity := gRecCfg.active.Rec.FeedVelocity;
	AxisPar.Acceleration := gRecCfg.active.Cfg.Creaser.FeedAxisAccel;
	AxisPar.Deceleration := gRecCfg.active.Cfg.Creaser.FeedAxisDecel;

	AxisControl.MoveVelocity := TRUE;
	AxisControl.MoveAbsolute := FALSE;
	AxisControl.MoveAdditive := FALSE;
	AxisControl.Stop := FALSE;
	AxisControl;
END_ACTION
```

#### Action_Move_Section_Distance.st
```iecst
ACTION Action_Move_Section_Distance:

	AxisControl.MoveAbsolute := FALSE;
	AxisControl.MoveAdditive := FALSE;
	AxisControl.MoveVelocity := FALSE;
	AxisControl.Stop := FALSE;
	AxisControl();

	AxisPar.Acceleration := gRecCfg.active.Cfg.Creaser.FeedAxisAccel;
	AxisPar.Deceleration := gRecCfg.active.Cfg.Creaser.FeedAxisDecel;
	AxisPar.Distance := 	gRecCfg.active.Rec.Crease.CreaseDistance_mm[ii_crease_count];
	AxisPar.Velocity := gRecCfg.active.Rec.FeedVelocity;

	AxisControl.MoveAdditive := TRUE;
	AxisControl();

END_ACTION
```

#### Action_Creaser_Idx.st
```iecst
ACTION Action_Creaser_Idx:
	setFlagCreaserIdxFinished := FALSE;

	IF setflagCreaserIndexCommand THEN
		setFlagTravelEdgeOffset := FALSE;
		setFlagCreaserWaitEdge := TRUE;
	END_IF;

	IF setFlagCreaserWaitEdge THEN
		IO.oCreaserCCWRotation := (gRecCfg.active.Rec.Crease.CreaserDirection = 0);
		IO.oCreaserCWRotation  := (gRecCfg.active.Rec.Crease.CreaserDirection = 1);

		IF setFlagTravelEdgeOffset AND bgTimerIsTimeOut(Timer_Creaser_Idx_Edge) THEN
			setFlagTravelEdgeOffset := FALSE;
			setFlagCreaserWaitEdge := FALSE;
			setFlagCreaserIdxFinished := TRUE;
		END_IF;

		CASE gRecCfg.active.Rec.Crease.ShaftSensorEdge OF
			0:
				IF IO.iCreaserShaftSensor AND NOT IO_LastCycle.iCreaserShaftSensor AND NOT setFlagTravelEdgeOffset THEN
					setFlagTravelEdgeOffset := TRUE;
					bgTimerStart(Timer_Creaser_Idx_Edge, Tms(gRecCfg.active.Rec.Crease.CreaserMotorIdxLag_S));
				END_IF;
			1:
				IF NOT IO.iCreaserShaftSensor AND IO_LastCycle.iCreaserShaftSensor AND NOT setFlagTravelEdgeOffset THEN
					setFlagTravelEdgeOffset := TRUE;
					bgTimerStart(Timer_Creaser_Idx_Edge, Tms(gRecCfg.active.Rec.Crease.CreaserMotorIdxLag_S));
				END_IF;
		END_CASE;
	ELSE
		IO.oCreaserCCWRotation := FALSE;
		IO.oCreaserCWRotation  := FALSE;
	END_IF;

	bgTimerCyclic(Timer_Creaser_Idx_Edge);

	setflagCreaserIndexCommand := FALSE;
END_ACTION
```

#### Action_AxisControl_Mgmt.st
```iecst
ACTION Action_AxisControl_Mgmt:

	IF EDGEPOS(iMachineErrorReset) THEN
		AxisControl.ErrorReset := TRUE;
	ELSIF EDGENEG(iMachineErrorReset)  THEN
		AxisControl.ErrorReset := FALSE;
	END_IF;

	IF AxisControl.ErrorReset AND NOT AxisControl.Error THEN //FBK errors only reset on + edge of error reset signal -> Clear reset signal when there are no errors!
		AxisControl.ErrorReset := FALSE;
	END_IF;

	Axis1; //Reference the PV cyclically to ensure it registers as being included in the program!
	AxisControl();//Call the function block responsible for executing the axis commands
END_ACTION
```

#### Action_Tally_Board_L.st
```iecst
ACTION Action_Tally_Board_L:

	RollerPos_ThisCycle := LREAL_TO_REAL(AxisControl.Position);

//	IF LREAL_TO_REAL(AxisControl.Position) > LREAL_TO_REAL(AxisControl_LastCycle.Position) THEN
//		delta_Board_Position := LREAL_TO_REAL(AxisControl.Position) - LREAL_TO_REAL(AxisControl_LastCycle.Position);
//	ELSE
//		IF (LREAL_TO_REAL(AxisControl_LastCycle.Position) > (0.99 * DEFINE_MM_ROLLER_REV)) AND (LREAL_TO_REAL(AxisControl.Position) < (1.01 * DEFINE_MM_ROLLER_REV)) THEN //Rollover
//			delta_Board_Position := (DEFINE_MM_ROLLER_REV - LREAL_TO_REAL(AxisControl_LastCycle.Position)) + LREAL_TO_REAL(AxisControl.Position);
//		ELSE
//			delta_Board_Position := LREAL_TO_REAL(AxisControl.Position) - LREAL_TO_REAL(AxisControl_LastCycle.Position);
//		END_IF;
	//	END_IF;
	delta_Board_Position := RollerPos_ThisCycle - RollerPos_LastCycle;

	Current_Board_Position := Current_Board_Position + delta_Board_Position;

	RollerPos_LastCycle := RollerPos_ThisCycle;
END_ACTION
```

#### Action_Validate_Board_Length.st
```iecst
ACTION Action_Validate_Board_Length:

	length_calculated_total := 0;
	flagBoardLengthCfgErr := FALSE;

	FOR ii_crease_count := 0 TO gRecCfg.active.Rec.Crease.CreaseCount - 1 BY 1 DO

		length_calculated_total := length_calculated_total + gRecCfg.active.Rec.Crease.CreaseDistance_mm[ii_crease_count] + gRecCfg.active.Rec.Crease.CreaseWidth_mm;

	END_FOR;

	IF length_calculated_total > (gRecCfg.active.Rec.Crease.TotalBoardLength + gRecCfg.active.Cfg.Creaser.BoardLengthTolerance) THEN
		gAlarms.Board_Length_GT_Confgd_Amount := TRUE;
		flagBoardLengthCfgErr := TRUE;
	ELSIF length_calculated_total < (gRecCfg.active.Rec.Crease.TotalBoardLength - gRecCfg.active.Cfg.Creaser.BoardLengthTolerance) THEN
		gAlarms.Board_Length_LT_Confgd_Amount := TRUE;
		flagBoardLengthCfgErr := TRUE;
	END_IF;

END_ACTION
```

#### Action_Eval_ErrorState_Statuses.st
```iecst
ACTION Action_Eval_ErrorState_Statuses:

	IF (MachineState <> MACHINE_STATE_ERROR AND MachineState <> MACHINE_STATE_INIT) THEN
		IF (NOT IO.iSafeMachineState) THEN //E-stop pressed
			gAlarms.Error_State_Unsafe_Machine := TRUE;
			MachineState := MACHINE_STATE_ERROR;
		ELSIF gAlarms.SM1_Disabled THEN //IO power disabled
			gAlarms.Error_State_SM1_Power := TRUE;
			MachineState := MACHINE_STATE_ERROR;
		ELSIF AxisControl.Error THEN //Servo Drive error
			gAlarms.Feed_Axis_Motor_Error := TRUE;
			MachineState := MACHINE_STATE_ERROR;
		ELSIF ProcessState = PRCS_STATE_ERROR THEN //Process Error
			gAlarms.Error_State_Process_Error := TRUE;
			MachineState := MACHINE_STATE_ERROR;
		ELSIF gRecCfg.active.Rec.Crease.CreaseCount > MAX_IDX_CREASES THEN //Configured crease amount error (shouldn't ever happen! PV tables shouldn't allow this, redundant here)
			gAlarms.Crease_Count_Greater_Max := TRUE;
			MachineState := MACHINE_STATE_ERROR;
		ELSIF NOT (gRecCfg.IO.Rec.O.Initial_Load = 1) THEN //Don't allow machine to run until you've loaded an inital recipe!
			gAlarms.Load_Recipe := TRUE;
			MachineState := MACHINE_STATE_ERROR;
		END_IF;
	END_IF;

END_ACTION
```

### Library Logical/Application/Master/libAS52XX

#### Application_Rec_Config.typ
```iecst
(*Insert your comment here.*)
(*Insert your comment here.*)

TYPE
	HMI_Trend_Limit_Par_typ : 	STRUCT
		Min : REAL;
		Max : REAL;
	END_STRUCT;
	Generic_Cfg_HMI_typ : 	STRUCT
		passwordSetup : STRING[15];
		passwordEngineer : STRING[15];
		passwordFactory : STRING[15];
		LoginTO_S : REAL;
		MachineLang : UDINT;
	END_STRUCT;
END_TYPE

(*Insert your comment here.*)
```

#### libAS52XX.fun
```iecst
FUNCTION_BLOCK FLASH
	VAR_INPUT
		TimeOn : TIME;
		TimeOff : TIME;
	END_VAR
	VAR_OUTPUT
		bFlashOut : BOOL;
	END_VAR
	VAR
		bFlashTrig : BOOL;
		TP_FLASH : TP;
		MaxTime : TIME;
	END_VAR
END_FUNCTION_BLOCK
```

#### FLASH.st
```iecst
(********************************************************************
 * COPYRIGHT -- Microsoft
 ********************************************************************
 * Library: Hernon
 * File: FLASH.st
 * Author: Rocky Hafen
 * Created: March 18, 2015
 ********************************************************************
 * Implementation of library Hernon
 ********************************************************************)

(* Flashes a BOOL output on/Off based on the inputs OnTime and OffTime *)
FUNCTION_BLOCK FLASH

	MaxTime := TimeOn + TimeOff ;
	TP_FLASH(IN:=bFlashTrig, PT:= (MaxTime + T#100ms));
	IF NOT bFlashTrig THEN
		bFlashTrig := TRUE;
	END_IF;

	IF (TP_FLASH.ET < TimeOn) THEN
		bFlashOut := TRUE;
	ELSIF (TP_FLASH.ET >= TimeOn) AND (TP_FLASH.ET <= MaxTime) THEN
		bFlashOut := FALSE;

	ELSE
		bFlashTrig := FALSE;
	END_IF;

END_FUNCTION_BLOCK
```

### Program Logical/Auxiliary_Services_Control/File_Handling

#### Init.st
```iecst
PROGRAM _INIT
	File_Manager_Control.MpLink := ADR(File_Manager_MpLink);
	File_Manager_Control.Enable := TRUE;
	File_Manager_Control.UIConnect := ADR(File_Manager_UIConnect);

	File_Manager_UIConnect.DeviceList.DeviceNames[0] := 'ROOT';
	File_Manager_UIConnect.DeviceList.DeviceNames[1] := 'Config';
	File_Manager_UIConnect.DeviceList.DeviceNames[2] := 'Recipe';
	File_Manager_UIConnect.DeviceList.DeviceNames[3] := '';
	File_Manager_UIConnect.DeviceList.DeviceNames[4] := '';
	File_Manager_UIConnect.DeviceList.DeviceNames[5] := '';

	File_Manager_Control.UISetup.FileListSize := 8;
	File_Manager_Control.UISetup.FileListScrollWindow := 5;

	File_Manager_Control;

	Alarm_File_UI.MpLink := ADR(File_Manager_MpLink);
	Alarm_File_UI.Enable := TRUE;
	Alarm_File_UI.Mode := mpALARM_BASIC_UI_MODE_ALL;

	Alarm_File_UI.UISetup.ImageSize := 20;
	Alarm_File_UI.UISetup.AlarmImage := ADR(Alarm_File.AlarmImage[0]);
	Alarm_File_UI.UISetup.AcknowledgeImage := ADR(Alarm_File.AcknowledgeImage[0]);
	Alarm_File_UI.UISetup.AddInfoStringSize := 100;
	Alarm_File_UI.UISetup.AddInfo := ADR(Alarm_File.AddInfo[0]);

	Alarm_File;
	Alarm_File_UI();

END_PROGRAM
```

### Program Logical/Auxiliary_Services_Control/Recipe_Handling

#### Types.typ
```iecst
TYPE
	Recipe_Cmd_local_typ : 	STRUCT
		Copy_default_to_save : BOOL;
		Copy_default_to_active : BOOL;
		Copy_save_to_active : BOOL;
		Copy_save_to_default : BOOL;
		Copy_active_to_save : BOOL;
		Copy_active_to_default : BOOL;
		Copy_internal_to_default : BOOL;
	END_STRUCT;
	Recipe_Status_local_typ : 	STRUCT
		save_differs_from_active : USINT;
		default_differs_from_save : USINT;
		active_differs_from_default : USINT;
	END_STRUCT;
	HMI_Rec_Command_Button_typ : 	STRUCT
		DP : USINT;
		Status : USINT;
		Lock : USINT;
	END_STRUCT;
	Recipe_HMI_Command_typ : 	STRUCT
		Refresh : HMI_Rec_Command_Button_typ;
		Save : HMI_Rec_Command_Button_typ;
		Load : HMI_Rec_Command_Button_typ;
		Delete : HMI_Rec_Command_Button_typ;
		Overwrite : HMI_Rec_Command_Button_typ;
		Copy : HMI_Rec_Command_Button_typ;
	END_STRUCT;
	Recipe_Config_local_struct : 	STRUCT
		cmd : Recipe_Cmd_local_typ;
		status : Recipe_Status_local_typ;
		HMI : Recipe_HMI_Command_typ;
	END_STRUCT;
	Recipe_loc_typ : 	STRUCT
		Cfg : Recipe_Config_local_struct;
		Rec : Recipe_Config_local_struct;
	END_STRUCT;
END_TYPE
```

#### Init.st
```iecst
PROGRAM _INIT
	IF gRecCfg.active.Cfg.MagicPrefix <> DEFINE_CONSTANT_MAGIC_PREFIX OR gRecCfg.save.Cfg.MagicPrefix <> DEFINE_CONSTANT_MAGIC_PREFIX OR gRecCfg.defaultvals.Cfg.MagicPrefix <> DEFINE_CONSTANT_MAGIC_PREFIX
		OR gRecCfg.active.Cfg.MagicSuffix <> DEFINE_CONSTANT_MAGIC_SUFFIX OR gRecCfg.save.Cfg.MagicSuffix <> DEFINE_CONSTANT_MAGIC_SUFFIX OR gRecCfg.defaultvals.Cfg.MagicSuffix <> DEFINE_CONSTANT_MAGIC_SUFFIX
		OR gRecCfg.active.Rec.MagicPrefix <> DEFINE_CONSTANT_MAGIC_PREFIX OR gRecCfg.save.Rec.MagicPrefix <> DEFINE_CONSTANT_MAGIC_PREFIX OR gRecCfg.defaultvals.Rec.MagicPrefix <> DEFINE_CONSTANT_MAGIC_PREFIX
		OR gRecCfg.active.Rec.MagicSuffix <> DEFINE_CONSTANT_MAGIC_SUFFIX OR gRecCfg.save.Rec.MagicSuffix <> DEFINE_CONSTANT_MAGIC_SUFFIX OR gRecCfg.defaultvals.Rec.MagicSuffix <> DEFINE_CONSTANT_MAGIC_SUFFIX
		THEN

		brsmemset(ADR(gRecCfg.defaultvals.Cfg), 0, SIZEOF(Global_Cfg_typ));
		brsmemset(ADR(gRecCfg.save.Cfg), 0, SIZEOF(Global_Cfg_typ));
		brsmemset(ADR(gRecCfg.active.Cfg), 0, SIZEOF(Global_Cfg_typ));

		brsmemset(ADR(gRecCfg.defaultvals.Rec), 0, SIZEOF(Global_Rec_typ));
		brsmemset(ADR(gRecCfg.save.Rec), 0, SIZEOF(Global_Rec_typ));
		brsmemset(ADR(gRecCfg.active.Rec), 0, SIZEOF(Global_Rec_typ));

		gRecCfg.active.Cfg.MagicPrefix := DEFINE_CONSTANT_MAGIC_PREFIX;
		gRecCfg.save.Cfg.MagicPrefix:= DEFINE_CONSTANT_MAGIC_PREFIX;
		gRecCfg.defaultvals.Cfg.MagicPrefix:= DEFINE_CONSTANT_MAGIC_PREFIX;

		gRecCfg.active.Cfg.MagicSuffix := DEFINE_CONSTANT_MAGIC_SUFFIX;
		gRecCfg.save.Cfg.MagicSuffix:= DEFINE_CONSTANT_MAGIC_SUFFIX;
		gRecCfg.defaultvals.Cfg.MagicSuffix:= DEFINE_CONSTANT_MAGIC_SUFFIX;

		gRecCfg.active.Rec.MagicPrefix := DEFINE_CONSTANT_MAGIC_PREFIX;
		gRecCfg.save.Rec.MagicPrefix:= DEFINE_CONSTANT_MAGIC_PREFIX;
		gRecCfg.defaultvals.Rec.MagicPrefix:= DEFINE_CONSTANT_MAGIC_PREFIX;

		gRecCfg.active.Rec.MagicSuffix := DEFINE_CONSTANT_MAGIC_SUFFIX;
		gRecCfg.save.Rec.MagicSuffix:= DEFINE_CONSTANT_MAGIC_SUFFIX;
		gRecCfg.defaultvals.Rec.MagicSuffix:= DEFINE_CONSTANT_MAGIC_SUFFIX;

		Set_Default_Config_Values(pCfg := ADR(gRecCfg.defaultvals.Cfg));
		Set_Default_Config_Values(pCfg := ADR(gRecCfg.save.Cfg));
		Set_Default_Config_Values(pCfg := ADR(gRecCfg.active.Cfg));

		gConfigName := 'No Config';

		Set_Default_Recipe_Values(pRec := ADR(gRecCfg.defaultvals.Rec));
		Set_Default_Recipe_Values(pRec := ADR(gRecCfg.save.Rec));
		Set_Default_Recipe_Values(pRec := ADR(gRecCfg.active.Rec));

		gRecipeName := 'No Recipe';

//		gAlarms.RecCfg.Default_Rec_Set := TRUE;

//		gAlarms.RecCfg.Default_Cfg_Set := TRUE;

//		SYSreset(1, 1);
	END_IF;

	gRecCfg.IO.Rec.I.FileName := 'rec1';
	gRecCfg.IO.Cfg.I.FileName := 'cfg1';

	Recipe_CSV_Control.MpLink := ADR(Recipe_CSV_MpLink);
	Recipe_CSV_Control.Enable := TRUE;
	Recipe_CSV_Control.DeviceName := ADR('Recipe');
	Recipe_CSV_Control.FileName := ADR(gRecCfg.IO.Rec.I.FileName);
	Recipe_CSV_Control.Category := ADR('Recipe');
	Recipe_CSV_Control.Header := ADR(Recipe_CSV_Header);

	Config_CSV_Control.MpLink := ADR(Config_CSV_MpLink);
	Config_CSV_Control.Enable := TRUE;
	Config_CSV_Control.DeviceName := ADR('Config');
	Config_CSV_Control.FileName := ADR(gRecCfg.IO.Cfg.I.FileName);
	Config_CSV_Control.Category := ADR('Config');
	Config_CSV_Control.Header := ADR(Config_CSV_Header);

	Recipe_CSV_RegPar.MpLink := ADR(Recipe_CSV_MpLink);
	Recipe_CSV_RegPar.Enable := TRUE;
	Recipe_CSV_RegPar.PVName := ADR('gRecCfg.save.Rec');
	Recipe_CSV_RegPar.Category := ADR('Recipe');

	Config_CSV_RegPar.MpLink := ADR(Config_CSV_MpLink);
	Config_CSV_RegPar.Enable := TRUE;
	Config_CSV_RegPar.PVName := ADR('gRecCfg.save.Cfg');
	Config_CSV_RegPar.Category := ADR('Config');

	Recipe_CSV_UI.MpLink := ADR(Recipe_CSV_MpLink);
	Recipe_CSV_UI.Enable := TRUE;
	Recipe_CSV_UI.UIConnect := ADR(gRecipe_CSV_UIConnect);

	Config_CSV_UI.MpLink := ADR(Config_CSV_MpLink);
	Config_CSV_UI.Enable := TRUE;
	Config_CSV_UI.UIConnect := ADR(gConfig_CSV_UIConnect);

	Recipe_CSV_UI.UISetup.RecipeListSize := 20;
	Recipe_CSV_UI.UISetup.RecipeListScrollWindow := 1;
	Recipe_CSV_UI.UISetup.Confirmation.RecipeCreate := TRUE;
	Recipe_CSV_UI.UISetup.Confirmation.RecipeLoad := TRUE;
	Recipe_CSV_UI.UISetup.Confirmation.RecipeSave := TRUE;
	Recipe_CSV_UI.UISetup.Confirmation.RecipeDelete := TRUE;

	Config_CSV_UI.UISetup.RecipeListSize := 20;
	Config_CSV_UI.UISetup.RecipeListScrollWindow := 1;
	Config_CSV_UI.UISetup.Confirmation.RecipeCreate := TRUE;
	Config_CSV_UI.UISetup.Confirmation.RecipeLoad := TRUE;
	Config_CSV_UI.UISetup.Confirmation.RecipeSave := TRUE;
	Config_CSV_UI.UISetup.Confirmation.RecipeDelete := TRUE;

	pRecCfgUIConnect ACCESS ADR(gRecipe_CSV_UIConnect);
	pCmd ACCESS ADR(loc.Rec.HMI);

	gRecipe_CSV_UIConnect.New.FileName := 'Rec_Name';
	gConfig_CSV_UIConnect.New.FileName := 'Cfg_Name';

	Recipe_CSV_Control;
	Recipe_CSV_RegPar;
	Recipe_CSV_UI;

	Config_CSV_Control;
	Config_CSV_RegPar;
	Config_CSV_UI;

	Alarm_Recipe_UI.MpLink := ADR(Recipe_CSV_MpLink);
	Alarm_Recipe_UI.Enable := TRUE;
	Alarm_Recipe_UI.Mode := mpALARM_BASIC_UI_MODE_ALL;

	Alarm_Recipe_UI.UISetup.ImageSize := 20;
	Alarm_Recipe_UI.UISetup.AlarmImage := ADR(Alarm_Recipe.AlarmImage[0]);
	Alarm_Recipe_UI.UISetup.AcknowledgeImage := ADR(Alarm_Recipe.AcknowledgeImage[0]);
	Alarm_Recipe_UI.UISetup.AddInfoStringSize := 100;
	Alarm_Recipe_UI.UISetup.AddInfo := ADR(Alarm_Recipe.AddInfo[0]);

	Alarm_Recipe;
	Alarm_Recipe_UI();

	Alarm_Config_UI.MpLink := ADR(Config_CSV_MpLink);
	Alarm_Config_UI.Enable := TRUE;
	Alarm_Config_UI.Mode := mpALARM_BASIC_UI_MODE_ALL;

	Alarm_Config_UI.UISetup.ImageSize := 20;
	Alarm_Config_UI.UISetup.AlarmImage := ADR(Alarm_Config.AlarmImage[0]);
	Alarm_Config_UI.UISetup.AcknowledgeImage := ADR(Alarm_Config.AcknowledgeImage[0]);
	Alarm_Config_UI.UISetup.AddInfoStringSize := 100;
	Alarm_Config_UI.UISetup.AddInfo := ADR(Alarm_Config.AddInfo[0]);

	Alarm_Config;
	Alarm_Config_UI();
END_PROGRAM
```

#### Set_Default_Config_Values.st
```iecst
FUNCTION Set_Default_Config_Values

	pCfg.HMI.passwordSetup := '1111';
	pCfg.HMI.passwordEngineer := '2222';
	pCfg.HMI.passwordFactory := '3333';

	Set_Default_Config_Values := 0;
END_FUNCTION
```

#### Set_Default_Recipe_Values.st
```iecst
FUNCTION Set_Default_Recipe_Values

	Set_Default_Recipe_Values := 0;
END_FUNCTION
```
